// TwinCAT 3 PLC project PlcProject
// Title: Boikon Template
// Company: Boikon
// ProjectVersion: 0.7.1.0000
// ProgramVersion: 3.1.4026.23
// CompilerDefines: IsTemplate
// libraries:
//   [Boikon Library], * (Boikon)
//   CmpBitmapPool, * (System)
//   VisuDialogs, * (System)
//   VisuDialogs
// project tree:
//   / CHECKBOUNDS.TcPOU (excluded from build), GlobalTextList.TcGTLO, ImagePool.TcIPO (not stored), VisualizationManager.TcVMO (not stored)
//   DevelopmentPlayground/MurrModLight60/ cntrl_MurrModLight60.TcPOU, MurrModLight60_IO.TcDUT, eMurrModLight60Colors.TcDUT, MurrModLight60_Outputs.TcDUT
//   DevelopmentPlayground/ObjectOrientedExamples/ IOopExmpl.TcIO (excluded from build), OopExmplBase.TcPOU (excluded from build), OopExmplExtension.TcPOU (excluded from build), OopExmplMain.TcPOU (excluded from build), OopExmplRandomObjectWithInterface.TcPOU (excluded from build)
//   DevelopmentPlayground/UnitTesting/ BreakLogging.TcPOU, Vis_Test.TcVIS
//   General/HMI/ HMI_ERR_General.TcDUT, HMI_General.TcPOU, HMI_MAN_General.TcDUT, HMI_SP_General.TcDUT, HMI_SP_GeneralShared.TcDUT (not stored), HMI_STS_General.TcDUT, HMI_WRN_General.TcDUT (not stored)
//   General/ utl_General.TcPOU, Vis_General.TcVIS
//   Main/ MAIN.TcPOU, PlcTask.TcTTO, VisGeneral.TcVIS, VisScmTemplate.TcVIS
//   Version/ Global_Version.TcGVL
//   _Control_Templates/cntrl_RbtFanuc/ cntrl_RbtFanucUnloadingRobot.TcPOU
//   _Control_Templates/cntrl_RbtFanuc/HMI/ HMI_ERR_RbtFanucUnloading.TcDUT, HMI_MAN_RbtFanucUnloading.TcDUT, HMI_RbtFanucUnloading.TcPOU, HMI_SP_RbtFanucUnloading.TcDUT, HMI_STS_RbtFanucUnloading.TcDUT, HMI_WRN_RbtFanucUnloading.TcDUT, Vis_RbtFanucUnloading.TcVIS
//   _Control_Templates/cntrl_RbtFanuc/LinkedIO/ RbtFanucUnloading_DataIn.TcDUT, RbtFanucUnloading_DataOut.TcDUT
//   _Control_Templates/cntrl_RbtFanuc/LinkedIO/Helpers/ RbtFanucUnloading_Array8Uint.TcDUT, RbtFanucUnloading_DataIn_Grouped.TcDUT, RbtFanucUnloadingt_DataOut_Grouped.TcDUT, RbtFanucUnloading_DI.TcDUT, RbtFanucUnloading_DO.TcDUT, RbtFanucUnloading_GI.TcDUT, RbtFanucUnloading_GO.TcDUT
//   _Control_Templates/cntrl_SafetyController/ cntrl_SafetyController1.TcPOU, HMI_ERR_SafetyController1.TcDUT (not stored), HMI_SafetyController1.TcPOU, HMI_STS_SafetyController1.TcDUT (not stored), HMI_WRN_SafetyController1.TcDUT, Vis_SafetyZone1.TcVIS
//   _Control_Templates/ utl_SignalColumn.TcPOU
//   _Globals/ eLogGroupsProject.TcDUT, Glbl.TcGVL, Glcn.TcGVL
//   _Scam/SCM_TemplateClean/EnumsAndState/ eTpc.TcDUT, sTpc.TcPOU
//   _Scam/SCM_TemplateClean/HMI/ HMI_ERR_TemplateClean.TcDUT, HMI_MAN_TemplateClean.TcDUT, HMI_SP_TemplateClean.TcDUT, HMI_STS_TemplateClean.TcDUT, HMI_TemplateClean.TcPOU (not stored), HMI_WRN_TemplateClean.TcDUT (not stored)
//   _Scam/SCM_TemplateClean/ SCM_TemplateClean.TcPOU
//   _Scam/SCM_TemplateMachinePart/EnumsAndState/ eTMP.TcDUT, sTmp.TcPOU
//   _Scam/SCM_TemplateMachinePart/HMI/ HMI_ERR_TemplateMachinePart.TcDUT, HMI_MAN_TemplateMachinePart.TcDUT, HMI_SP_TemplateMachinePart.TcDUT (not stored), HMI_STS_TemplateMachinePart.TcDUT (not stored), HMI_TemplateMachinePart.TcPOU, HMI_WRN_TemplateMachinePart.TcDUT
//   _Scam/SCM_TemplateMachinePart/ SCM_TemplateMachinePart.TcPOU

CONFIGURATION PlcProject
    RESOURCE PLC ON TwinCAT3
        TASK PlcTask(INTERVAL := T#1ms, PRIORITY := 6);
        PROGRAM MAIN WITH PlcTask : MAIN;
    END_RESOURCE
END_CONFIGURATION

// ---- DevelopmentPlayground/MurrModLight60/MurrModLight60_IO.TcDUT
//ignore unused variables
{attribute 'analysis' := '-33'}
TYPE MurrModLight60_IO :
UNION
	//hw linking
	_Q AT %Q*: ARRAY[0..7] OF BYTE;
	//program use
	Control:MurrModLight60_Outputs;
END_UNION
END_TYPE

// ---- DevelopmentPlayground/MurrModLight60/eMurrModLight60Colors.TcDUT
{attribute 'qualified_only'}
{attribute 'strict'}
{attribute 'to_string'}
TYPE eMurrModLight60Colors :
(
	COLOR_OFF:= 		2#0,
	COLOR_RED:= 		2#001,
	COLOR_GREEN:= 		2#010,
	COLOR_YELLOW:= 		2#011,
	COLOR_BLUE:= 		2#100,
	COLOR_CUSTOM1:= 	2#101,
	COLOR_CUSTOM2:= 	2#110,
	COLOR_WHITE:= 		2#111,
	
	PAT_CONTINIOUS:= 	2#001000,
	PAT_BLINKING:=		2#010000,
	PAT_FLASHING:= 		2#011000,
	PAT_GRADBLINK:=		2#100000,
	
	SPD_LOW:=			2#01000000,
	SPD_MID:=			2#10000000,
	SPD_FAST:=			2#11000000
)BYTE;
END_TYPE

// ---- DevelopmentPlayground/MurrModLight60/MurrModLight60_Outputs.TcDUT
//ignore unused variables
{attribute 'analysis' := '-33'}
TYPE MurrModLight60_Outputs :
STRUCT
	//byte 0
	Stack1:BYTE; //combined bits for stack settings (color/pat/speed)
	//byte 1
	Stack2:BYTE; //combined bits for stack settings (color/pat/speed)
	//byte 2
	Stack3:BYTE; //combined bits for stack settings (color/pat/speed)
	
	//byte 3-4
	SpareByte3:BYTE;
	SpareByte4:BYTE;
	
	//byte 3
	BuzzerOnOff:BIT;
	BuzzerTypeBit0:BIT;
	BuzzerTypeBit1:BIT;
	BuzzerTypeBit2:BIT;

	BuzzerLoudnessBit0:BIT;
	BuzzerLoudnessBit1:BIT;
	BuzzerLoudnessBit2:BIT;
	BuzzerLoudnessBit3:BIT;
	
	//byte 4
	StackMode:BIT;
	LevelMode:BIT;
	SliceMode:BIT;
	SpareByte4_3:BIT;
	SyncModeAct:BIT;
	SyncModeTrig:BIT;
	UserPrefSelBit0:BIT;
	UserPrefSelBit1:BIT;
	
	//byte 5
	TopDown:BIT;
	SpareBYte5_1:BIT;
	ColorDom:BIT;
	EcoMode:BIT;
	SpareByte5_4:BIT;
	
	StacksBit0:BIT;		
	StacksBit1:BIT;
	StacksBit2:BIT;
END_STRUCT
END_TYPE

// ---- General/HMI/HMI_ERR_General.TcDUT
TYPE HMI_ERR_General :
STRUCT
	//General IO
	//prio's: emergency stop items == 100, e-circuit=99, default (nothing specified) = 50
	//adjust as needed
	ExampleErrorPreConfiggedPrio:BOOL;					//Error[prio=90] Example error with preconfigured prio (key only used at first creation/adding to the HMI-alarm-list-file)
END_STRUCT
END_TYPE

// ---- General/HMI/HMI_MAN_General.TcDUT
TYPE HMI_MAN_General :
STRUCT
	//note: manuals are normally used for controls, not for general
	//PB_MyManualCommand:bool;
END_STRUCT
END_TYPE

// ---- General/HMI/HMI_SP_General.TcDUT
TYPE HMI_SP_General :
STRUCT
	{warning 'TODO Template: example / remove when not needed'}
	//These setpoint are made available for all blocks
	Shared:HMI_SP_GeneralShared;											//Common setpoints used for multiple machine parts
END_STRUCT
END_TYPE

// ---- General/HMI/HMI_STS_General.TcDUT
TYPE HMI_STS_General :
STRUCT
	Version:STRING(23);								//Project version
END_STRUCT
END_TYPE

// ---- _Control_Templates/cntrl_RbtFanuc/HMI/HMI_ERR_RbtFanucUnloading.TcDUT
TYPE HMI_ERR_RbtFanucUnloading EXTENDS HMI_ERR_RbtFanuc:
STRUCT
	;//add custom bools on top of library block here
END_STRUCT
END_TYPE

// ---- _Control_Templates/cntrl_RbtFanuc/HMI/HMI_MAN_RbtFanucUnloading.TcDUT
TYPE HMI_MAN_RbtFanucUnloading EXTENDS HMI_MAN_RbtFanuc:
STRUCT
	;//add custom bools on top of library block here
END_STRUCT
END_TYPE

// ---- _Control_Templates/cntrl_RbtFanuc/HMI/HMI_SP_RbtFanucUnloading.TcDUT
TYPE HMI_SP_RbtFanucUnloading EXTENDS HMI_SP_RbtFanuc:
STRUCT
	;//add custom on top of library block here
END_STRUCT
END_TYPE

// ---- _Control_Templates/cntrl_RbtFanuc/HMI/HMI_STS_RbtFanucUnloading.TcDUT
TYPE HMI_STS_RbtFanucUnloading EXTENDS HMI_STS_RbtFanuc:
STRUCT
	;//add custom on top of library block here
END_STRUCT
END_TYPE

// ---- _Control_Templates/cntrl_RbtFanuc/HMI/HMI_WRN_RbtFanucUnloading.TcDUT
TYPE HMI_WRN_RbtFanucUnloading EXTENDS HMI_WRN_RbtFanuc:
STRUCT
	;//add custom bools on top of library block here
END_STRUCT
END_TYPE

// ---- _Control_Templates/cntrl_RbtFanuc/LinkedIO/RbtFanucUnloading_DataIn.TcDUT
{attribute 'analysis' := '-33'}
(*
	Plclinking:
		-Choose variable: ByAddress
			>
	Robot IO config:
		Go to config when you're in the DO/DI / UO/UI / GO/GI sections.
		if needed, delete default configs
		To link to ethercat card use, 
			rack 106 (some robot-types might use another rack nr. check manual) 
			slot 1
			start =>offset on the linked variables
			
		Example for this situation:
			UO => rack 106, slot 1, start 0   =>this will link UO[1]-CmdEnabled to ByAddress.0, which is good since Vars._UO.CmdEnabled is the first bit declared in the Vars structure.
			since the struct declared in the plc for the UO (Fanuc_StatusWord) is aligned to 3 bytes, DO must have an offset of 16
			DO => rack 106, slot 1, start 16 
*)
TYPE RbtFanucUnloading_DataIn :
UNION
	//linked directly to robot 
	ByAddress AT %I*: ARRAY[0..3] OF RbtFanucUnloading_Array8Uint;
	
	//data as variables for use in the plc
	Vars:RbtFanucUnloading_DataIn_Grouped;

END_UNION
END_TYPE

// ---- _Control_Templates/cntrl_RbtFanuc/LinkedIO/RbtFanucUnloading_DataOut.TcDUT
{attribute 'analysis' := '-33'}
(*
	Robot IO config:
		Go to config when you're in the DO/DI / UO/UI / GO/GI sections.
		if needed, delete default configs
		To link to ethercat card use, 
			rack 106 (some robot-types might use another rack nr. check manual) 
			slot 1
			start =>offset on the linked variables
			
		Example for this situation:
			UO => rack 106, slot 1, start 0   =>this will link UO[1]-CmdEnabled to ByAddress.0, which is good since Vars._UO.CmdEnabled is the first bit declared in the Vars structure.
			since the struct declared in the plc for the UO (Fanuc_StatusWord) is aligned to 3 bytes, DO must have an offset of 16
			DO => rack 106, slot 1, start 16 
*)
TYPE RbtFanucUnloading_DataOut :
UNION
	//linked directly to robot 
	ByAddress AT %Q*: ARRAY[0..3] OF RbtFanucUnloading_Array8Uint;
	
	//data as variables for use in the plc
	Vars:RbtFanucUnloadingt_DataOut_Grouped;

END_UNION
END_TYPE

// ---- _Control_Templates/cntrl_RbtFanuc/LinkedIO/Helpers/RbtFanucUnloading_Array8Uint.TcDUT
{attribute 'analysis' := '-33'}
TYPE RbtFanucUnloading_Array8Uint :
STRUCT
	_E: ARRAY [0..7] OF UINT;
END_STRUCT
END_TYPE

// ---- _Control_Templates/cntrl_RbtFanuc/LinkedIO/Helpers/RbtFanucUnloading_DataIn_Grouped.TcDUT
{attribute 'pack_mode' := '1'} //no gaps! (compiler tries to allign with base types)
TYPE RbtFanucUnloading_DataIn_Grouped :
STRUCT
	_UO:RbtFanuc_StatusWord; 			//24bits	>>start pt=1
	_DO:RbtFanucUnloading_DO;			//32 bits	>>start pt=25
	_GO:RbtFanucUnloading_GO;			//16 bits	>>start pt=57
END_STRUCT
END_TYPE

// ---- _Control_Templates/cntrl_RbtFanuc/LinkedIO/Helpers/RbtFanucUnloadingt_DataOut_Grouped.TcDUT
{attribute 'pack_mode' := '1'} //no gaps! (compiler tries to allign with base types and might skip bits otherwise)
{attribute 'analysis' := '-33'}
TYPE RbtFanucUnloadingt_DataOut_Grouped :
STRUCT
	_UI:RbtFanuc_ControlWord;			//24bits	>>start pt=1
	_DI:RbtFanucUnloading_DI;			//32 bits	>>start pt=25
	_GI:RbtFanucUnloading_GI;			//16 bits	>>start pt=57
END_STRUCT
END_TYPE

// ---- _Control_Templates/cntrl_RbtFanuc/LinkedIO/Helpers/RbtFanucUnloading_DI.TcDUT
{attribute 'analysis' := '-33'}
TYPE RbtFanucUnloading_DI :
STRUCT
	//bits 0-15
	SN_InitLeft:BIT;		//DI+00 command init/start left side
	SN_InitRight:BIT;		//DI+01 command init/start left side
	SN_CylInOk:BIT;			//DI+02 command resp cylinder is in
	SN_CylOutOk:BIT;		//DI+03 command resp cylinder is out
	SN_CrateEmptyOk:BIT;	//DI+04 command resp crate is empty
	SN_RequestDumpOk:BIT;	//DI+05 command resp crate is dumped
	SN_PayloadConfirm:BIT;	//DI+-6 command to confirm payload > must be setup in dcs
	bit07:BIT;
	bit08:BIT;
	bit09:BIT;
	PC_Left_Z:BIT;			//DI+10
	PC_Right_Z:BIT;			//DI+11
	PX_Left_X:BIT;			//DI+12
	PX_Right_X:BIT;			//DI+13
	bit14:BIT;
    bit15:BIT;
    K_DropBasket:BIT;		//Command from scam to drop basket
    bit17:BIT;
    bit18:BIT;
    bit19:BIT;
    bit20:BIT;
    bit21:BIT;
    bit22:BIT;
    bit23:BIT;
    bit24:BIT;
    bit25:BIT;
    bit26:BIT;
    bit27:BIT;
    bit28:BIT;
    bit29:BIT;
    bit30:BIT;
    bit31:BIT;
END_STRUCT
END_TYPE

(*
	//copy to your project and adapt names + number of bits to your situation
	//bits 0-15
	bit00:BIT;
    bit01:BIT;
    bit02:BIT;
    bit03:BIT;
    bit04:BIT;
    bit05:BIT;
    bit06:BIT;
    bit07:BIT;
    bit08:BIT;
    bit09:BIT;
    bit10:BIT;
    bit11:BIT;
    bit12:BIT;
    bit13:BIT;
    bit14:BIT;
    bit15:BIT;
    bit16:BIT;
    bit17:BIT;
    bit18:BIT;
    bit19:BIT;
    bit20:BIT;
    bit21:BIT;
    bit22:BIT;
    bit23:BIT;
    bit24:BIT;
    bit25:BIT;
    bit26:BIT;
    bit27:BIT;
    bit28:BIT;
    bit29:BIT;
    bit30:BIT;
    bit31:BIT;
*)

// ---- _Control_Templates/cntrl_RbtFanuc/LinkedIO/Helpers/RbtFanucUnloading_DO.TcDUT
{attribute 'analysis' := '-33'}
TYPE RbtFanucUnloading_DO :
STRUCT
	//bits 0-15
	SN_InitLeftOk:BIT;		//DO+00 command init/start left side
	SN_InitRightOk:BIT;		//DO+01 command init/start left side
	SN_CylIn:BIT;			//DO+02 command cylinder is in
	SN_CylOut:BIT;			//DO+03 command cylinder is out
	SN_CrateEmpty:BIT;		//DO+04 command crate is empty
	SN_RequestDump:BIT;		//DO+05 command crate is dumped
    bit06:BIT;
    bit07:BIT;
    bit08:BIT;
	STS_Error:BIT;			//DO+09 status in error
    STS_Latched1:BIT;		//DO+10
    STS_Latched2:BIT;		//DO+11
    bit12:BIT;
    bit13:BIT;
    bit14:BIT;
    bit15:BIT;
	K_DropBasket_OK:BIT;	//Response from robot drop basket ok
    bit17:BIT;
    bit18:BIT;
    bit19:BIT;
    bit20:BIT;
    bit21:BIT;
    bit22:BIT;
    bit23:BIT;
    bit24:BIT;
    bit25:BIT;
    bit26:BIT;
    bit27:BIT;
    bit28:BIT;
    bit29:BIT;
    bit30:BIT;
    bit31:BIT;
END_STRUCT
END_TYPE


(*
bit00:BIT;
    bit01:BIT;
    bit02:BIT;
    bit03:BIT;
    bit04:BIT;
    bit05:BIT;
    bit06:BIT;
    bit07:BIT;
    bit08:BIT;
    bit09:BIT;
    bit10:BIT;
    bit11:BIT;
    bit12:BIT;
    bit13:BIT;
    bit14:BIT;
    bit15:BIT;
    bit16:BIT;
    bit17:BIT;
    bit18:BIT;
    bit19:BIT;
    bit20:BIT;
    bit21:BIT;
    bit22:BIT;
    bit23:BIT;
    bit24:BIT;
    bit25:BIT;
    bit26:BIT;
    bit27:BIT;
    bit28:BIT;
    bit29:BIT;
    bit30:BIT;
    bit31:BIT;
*)

// ---- _Control_Templates/cntrl_RbtFanuc/LinkedIO/Helpers/RbtFanucUnloading_GI.TcDUT
{attribute 'analysis' := '-33'}
TYPE RbtFanucUnloading_GI :
STRUCT
	//copy to your project and adapt names + number of bits to your situation
	Word0:WORD;
END_STRUCT
END_TYPE

// ---- _Control_Templates/cntrl_RbtFanuc/LinkedIO/Helpers/RbtFanucUnloading_GO.TcDUT
{attribute 'analysis' := '-33'}
TYPE RbtFanucUnloading_GO :
STRUCT
	//GO[1]
	ErrorNr:UINT;
	State:UINT;
	NrPickedCrates:UINT;
	NrPayload:uint;
END_STRUCT
END_TYPE

// ---- _Control_Templates/cntrl_SafetyController/HMI_WRN_SafetyController1.TcDUT
//Extend the base errors with project errors
TYPE HMI_WRN_SafetyController1 EXTENDS HMI_WRN_SafetyLogic:
STRUCT
	//note: errors for inputs moved to input-instances
	;
END_STRUCT
END_TYPE

// ---- _Globals/eLogGroupsProject.TcDUT
{attribute 'qualified_only'}
TYPE eLogGroupsProject :
(
	//the first 8 bits are taken/reserved for the boikon library groups: Boikon_Library.eLogGroups
	(*
	Off					:= 2#0,					//this channel will not get logged
	Default				:= 2#1,					//the library blocks will automaticly give the default group for the logged type, otherwise a custom group can be chosen
	Inputs				:= 2#10,	
	Outputs 			:= 2#100,
	Analogs				:= 2#1000,
	Cntrl_states		:= 2#10000,				//states for controls/utilities (servo blocks for example)
	*)
	//project groups, in total 32 bits available
	//add/rename/remove groups as needed
	SCM_States 			:=SHL(2#1,8),
	SCM_CommSignals		:=SHL(2#1,9),
	Spare				:=SHL(2#1,10),
	Template			:=SHL(2#1,11),
	TestServoPos		:=SHL(2#1,12)
)DWORD;
END_TYPE

//info on attributes:
//strict 			: also tests if the name is not used for something else
//to_string			: allows the enum to be converted to string
//qualified_only 	: forces the user to start witht the type name (to avoid the situation that accidentially another enum is used)

// ---- _Scam/SCM_TemplateClean/EnumsAndState/eTpc.TcDUT
//enum of states
{attribute 'strict'}
{attribute 'to_string'}
{attribute 'qualified_only'}
TYPE eTpc :
(
	//NOTE @ copy of this enum, adapt existing state names:
	Disabled := -1, //-1: to make sure the code for disabling fires
	TotalReset,
	Initialise,
	Rest
)INT;
END_TYPE

//info on attributes:
//strict 			: don't allow mixing of types
//to_string			: allows the enum to be converted to string
//qualified_only 	: forces the user to start witht the type name (to avoid the situation that accidentially another enum is used)

// ---- _Scam/SCM_TemplateClean/HMI/HMI_ERR_TemplateClean.TcDUT
TYPE HMI_ERR_TemplateClean :
STRUCT
	(*
		Rules:
		Errors shall only be off type BOOL
		Errors shall be set >> the HMI block will do the resetting

		Syntax convention:
		a clear variable name which describes the error			as described below
		InitNotEmpty:BOOL;										//Error [machinepart]: not empty during initialisation
		
		prio's: emergency stop items == 100, e-circuit=99, default (nothing specified) = 50
		adjust as needed
		//example how to pre-set error priorities for the HMI. Default errors get prio 50, Recommend prio 100 for e-stop buttons etc
		ExampleErrorPreConfiggedPrio:BOOL;					//Error[prio=90] Example error with preconfigured prio (key only used at first creation/adding to the HMI-alarm-list-file)
	*)
END_STRUCT
END_TYPE

// ---- _Scam/SCM_TemplateClean/HMI/HMI_MAN_TemplateClean.TcDUT
TYPE HMI_MAN_TemplateClean :
STRUCT

END_STRUCT
END_TYPE

// ---- _Scam/SCM_TemplateClean/HMI/HMI_SP_TemplateClean.TcDUT
TYPE HMI_SP_TemplateClean :
STRUCT
	MachinePartEnabled:BOOL:=TRUE;				//block is enabled >> can be used to disable part(s) of the machine
END_STRUCT
END_TYPE

// ---- _Scam/SCM_TemplateClean/HMI/HMI_STS_TemplateClean.TcDUT
TYPE HMI_STS_TemplateClean :
STRUCT
	IsEmpty:BOOL;												//Machinepart is empty
END_STRUCT
END_TYPE

// ---- _Scam/SCM_TemplateMachinePart/EnumsAndState/eTMP.TcDUT
//enum of states
{attribute 'strict'}
{attribute 'to_string'}
{attribute 'qualified_only'}
TYPE eTMP :
(
	TotalReset,
	InitCyl,
	InitSrv,
	InitCamQuickFocus,
	InitCamLoadJob,
	Rest,
	SrvPosStart,
	SrvPosStartInterl,
	SrvPosEnd,
	SrvPosEndIntrl,
	CylOut,
	CylIn,
	MtrStartFwd,
	MtrStop,
	MtrStartRev,
	CamReady,
	CamTrig,
	MultiStepTest2,
	MultiStepTest3,
	
	//Example how to use the organiser semi-automode
	//this is a special case in which the operator can choose with a button for example to let the machine do special things 
	//like put servos+clinders automated in a position for configuring/measuring
	
	SemiAutoStart,
	SemiAutoStop
);
END_TYPE

//info on attributes:
//strict 			: don't allow mixing of types
//to_string			: allows the enum to be converted to string
//qualified_only 	: forces the user to start witht the type name (to avoid the situation that accidentially another enum is used)

// ---- _Scam/SCM_TemplateMachinePart/HMI/HMI_ERR_TemplateMachinePart.TcDUT
TYPE HMI_ERR_TemplateMachinePart :
STRUCT
	(*
		Rules:
		Errors shall only be off type BOOL
		Errors shall be set >> the HMI block will do the resetting

		Syntax convention:
		a clear variable name which describes the error			as described below
		InitNotEmpty:BOOL;										//Error [machinepart]: not empty during initialisation
		
		prio's: emergency stop items == 100, e-circuit=99, default (nothing specified) = 50
		adjust as needed
		//example how to pre-set error priorities for the HMI. Default errors get prio 50, Recommend prio 100 for e-stop buttons etc
		ExampleAddPrioForHmiError:BOOL;					//Error[prio=90] TemplateMachinePart: we have an error!
	*)
	InitNotEmpty:BOOL;								//Error [machinepart]: not empty during initialisation
	
	//example how to pre-set error priorities for the HMI. Default errors get prio 50, Recommend prio 100 for e-stop buttons etc
	ExampleAddPrioForHmiError:BOOL;					//Error[prio=100] TemplateMachinePart: we have an error!
	
	//test log error by name, very long name, truncation
	TestStupidLongErrorNameWillItGetLoggedAbcdefghijklmnopqrstuvwzyzAbcdefghijklmnopqrstuvwzyzAbcdefghijklmnopqrstuvwzyzAbcdefghijklmnopqrstuvwzyzAbcdefghijklmnopqrstuvwzyz:BOOL;
END_STRUCT
END_TYPE

// ---- _Scam/SCM_TemplateMachinePart/HMI/HMI_MAN_TemplateMachinePart.TcDUT
TYPE HMI_MAN_TemplateMachinePart :
STRUCT
	;
END_STRUCT
END_TYPE

// ---- _Scam/SCM_TemplateMachinePart/HMI/HMI_WRN_TemplateMachinePart.TcDUT
TYPE HMI_WRN_TemplateMachinePart :
STRUCT
	(*
		Rules:
		Warnings shall only be of type BOOL
		Warnings can be set / reset / activated as you need it (unlike errors!). 
		
		Syntax convention:
		a clear variable name which describes the warning		as described below
		StepLockActive:BOOL;									//Warning [machinepart]: in step modus (steps are held until confirmation the continue to the next step)
	*)
	NotRdyRcv_Discharge:BOOL;								//Warning [machinepart]: not ready to receive products
	CameraNotReady:BOOL;									//Warning [machinepart]: waiting for camera ready
	PlanoBufferNeedsRefill:BOOL;							//Warning [machinepart]: Planobuffer needs refill
END_STRUCT
END_TYPE

// ---- Version/Global_Version.TcGVL
{attribute 'TcGenerated'}
{attribute 'no-analysis'}
{attribute 'linkalways'}
// This function has been automatically generated from the project information.
VAR_GLOBAL CONSTANT
	{attribute 'const_non_replaced'}
	stLibVersion_Boikon_Template : ST_LibVersion := (iMajor := 0, iMinor := 7, iBuild := 1, iRevision := 0, nFlags := 0, sVersion := '0.7.1.0');
END_VAR

// ---- _Globals/Glbl.TcGVL
//project related global variables
{attribute 'qualified_only'}
{attribute 'analysis' := '-33'}
VAR_GLOBAL
//Variables set by Checkbounds. This function increases processor load and should be disabled once bounds problems are solved
	OutOfBounds:BOOL:=FALSE;						//Should always be false otherwise a bounds problem >> function CHECKBOUNDS must be implemented in the project, check the beckhoff help !only for testing purposes!
	OutOfBoundsIndex:DINT := 0;						//Index trying to address which was out of bounds


(*Project*)
	//TODO TEMPLATE >>
		//adapt / remove as needed
	SimEnable:BOOL:=FALSE;					//Enable simulation (when false, all simulation setpoints will be set to false
	Sim_MyMachinePart:BOOL; 				//Simulate only a part of the machine (in this case the template example)
END_VAR
// {attribute 'qualified_only'} >>forces the user to add the DUT name in front of the variables
// {attribute 'analysis' := '-33'} >>deactivate error unused variable for next variable/struct

// ---- _Globals/Glcn.TcGVL
//project related global constants
{attribute 'qualified_only'}
VAR_GLOBAL CONSTANT

{info 'TODO: TEMPLATE REMOVE WHEN NOT NEEDED'}
//array sizes >> use this to initialise the array AND then use it in the for loops which run through the arrays etc
	//MaxIndexForMyArray:INT:=10;
	//to be used as:
	//MyArray: array[0..MaxIndexForMyArray] of bool;
	//and then
	//FOR index:=0 to MaxIndexForMyArray by 1 DO ...
END_VAR

// ---- DevelopmentPlayground/ObjectOrientedExamples/IOopExmpl.TcIO
(*An interface describes the must have methods for a functionblock
	-now you know for sure that a block implementing this interface will have the methods described here
*) 
INTERFACE IOopExmpl

METHOD MustHaveMethod : BOOL
VAR_INPUT
	I:BOOL;
END_VAR
END_METHOD

END_INTERFACE

// ---- Main/MAIN.TcPOU
(*Basic MAIN with an example organiser and scam*)
{info '_Welcome to the Boikon Twincat 3 Template'}
{info '__Please read the _Readme.txt for more info'}
{warning 'TODO Template: upload boot project at online change is disabled in project settings, RE-ENABLE!!!!'}
PROGRAM MAIN
VAR
	//General collection of system wide IO and control blocks
	General: Utl_General;

	//TODO TEMPLATE: here in the example only 1 organiser is used, add + rename as needed
	Organiser:cntrl_Organiser(						
		SP_TmrReset := T#1S,
		SP_TmrResetES := T#3S);
END_VAR

//TODO TEMPLATE >> Remove this section, it is for testing the library and template
//Also remove the define from here: project/properties/compile/compiler defines/IsTemplate
{IF defined (IsTemplate)}
	{warning 'TODO Template: testing is enabled >> Remove the define and clean all "TODO TEMPLATE" locations'}
	{attribute 'analysis' := '-33'}
	VAR
		//Scam-template >> use tool supplied in the folder, to make a copy for your own scam implementation 
		OrganiserFake: cntrl_OrganiserFake;
		
		//Fully functional test scam which uses almost all library blocks >> can be used as example how to do things 
		ExampleMachinePart: SCM_TemplateClean;

		//just to show it's possible
		//these variables will now have the same comment (these 2 lines)
		//*multiline comment still is a kind of broken in the editor, parts will dissapear..
		MyBool1,MyBool2,MyBool3:BOOL;  

		//Banner-Multicolor signal lamp
		//NOTE: You can use it this way for multiple organisers as well, just keep calling ..M_UpdateOrganiserState(xxx) for each organiser  
		LP_OrgGroupMachinePart:Cntrl_BannerKxx(
			Intensity:= eBannerKxx_Intensity.Low);

		LP_MurrTest: cntrl_MurrModLight60(NrOfStacks:=3);

		//Performance test	
		HM_ProfileBlocks:BOOL;
		StopWatchGeneral,StopWatchMachineStuff:profiler;
		
		//casting works with a lot of types, example time
		sMyUtcTime:string;

		//string value to int test
		sValue1,sValue2,sValue3:STRING := '123';
		sValue4,sValue5:string(1);
		b0Value:BYTE;
		iValue1,iValue2:INT;
		
		
		//random tests
		dbglreal:LREAL;
		dbgbool1,dbgbool2,dbgbool3:BOOL;
	END_VAR
{END_IF}

//TODO template: general actions can be added here. 
//in utl_General I've added the usual suspects needed for a machine.
//please keep in mind I've only included common reocurring items, you need to thoroughly check / update / clean the block!
a_General();
b_MachinePart();

ACTION a_General:
//General is the place for all in-/outputs not specific belonging to a machinepart like:
//	-handling of boikonlibrary functionality
//	-general start/stop/reset buttons + lights
//	-general airpressure sensor
//	-safety components: control + errors for doors/lightscreens/pushbuttons
//	-ethercat diagnostics
General(
	//Reset command + general start/stop/reset button lights > add organisers as needed, use OR
	I_SN_ResetErrors:= Organiser.Reset_K,
	I_SN_Lp_Pb_StartAll:= Organiser.Q_LP_Start,
	I_SN_Lp_Pb_StopAll:= Organiser.Q_LP_Stop,
	I_SN_Lp_Pb_ResetAll:= Organiser.Q_LP_Reset,
	
	//Machine status
	I_STS_Error:=,
	I_STS_NoDischarge:=,
	I_STS_OperatorInput:=,
	I_STS_Running:=,	
	
	//Organiser/SCAM control-outputs
	Q_SN_ES_Zone1_OK=>, 
	Q_SN_StartAll=>,
	Q_SN_StopAll=>,
	Q_SN_ResetAll=> ,
	Q_SN_TotalResetAll=>);

//TODO TEMPLATE remove if not needed
//Organiser(s) Banner multicolor indicator light
//	this is an example on how to use it to show the status of an organiser
//	1) you can also manually control the lamp with the given M_Set... methods, but then don't call M_UpdateOrganiserState anymore!
//	2) inside general would be a better place but there you can't access the Organiser instances easily (or you tresspass OOP by doing things like: main.Organiser inside.... > don't do that!)
LP_OrgGroupMachinePart.M_UpdateOrganiserState(Organiser); //call this method for each organiser belonging to this group
LP_OrgGroupMachinePart();

//TODO TEMPLATE remove banner break-time
//Mess around with the banner multicolor lamp >> if break-time, overwrite previous (organiser-state) call with a manual set color
IF(	(	BknGlbl.LocalSystemTime.wHour = 10
		AND_THEN BknGlbl.LocalSystemTime.wMinute <= 15)
	OR	(	BknGlbl.LocalSystemTime.wHour = 12
			AND_THEN BknGlbl.LocalSystemTime.wMinute >= 30)
	OR	(	BknGlbl.LocalSystemTime.wHour >= 17))
THEN
	LP_OrgGroupMachinePart.M_Set2ColorAnimation(
		I_Color1 := eBannerKxx_Color.Yellow,
		I_Color2 := eBannerKxx_Color.Red,
		I_Animation:= eBannerKxx_AnimationType.HalfHalfRotate,
		TRUE); 
	LP_OrgGroupMachinePart();
END_IF
END_ACTION

ACTION b_MachinePart:
//Note: if the machine consists of several machine parts with their own organiser then for a cleaner structure make a seperate action for each part
//todo think about this

Organiser(
	//Emergencystop zone for scams connected to this organiser
	I_SN_ES_OK:= General.Q_SN_ES_Zone1_OK,
	I_SN_ExternalError:= General.Q_SN_ERR_General, //organiser should go into error caused by external factors (like a general error)
	//Total reset command for this organiser and connected scams
	//note: scams that communicate with each other via interlocking should have the same total reset command otherwise deadlocks will occur!
	I_SN_TotalReset:= General.Q_SN_TotalResetAll,
	I_PB_Start:= General.Q_SN_StartAll,
	I_PB_Stop:= General.Q_SN_StopAll,
	I_PB_Reset:= General.Q_SN_ResetAll, 
	Q_LP_Start=>, 
	Q_LP_Stop=>, 
	Q_LP_Reset=>);

ExampleMachinePart( //todo remove true
	I_K_ES_OK:= General.Q_SN_ES_Zone1_OK, 			//Emergency stop for this zone OK. @ mutliple zones, fbGeneral must be adapted to supply these signals for each zone
	I_Organiser:= Organiser, 						//Control signals from the organiser
	I_STS_SUP_Empty:= , 							//Connect to upstream. The upstream is empty, use this to enter energy-save mode (stop conveyors etc)
	Q_STS_Empty=> , 								//Connect to downstream. The supply is empty and this part is now empty and in energy-save mode
	Q_SN_SUP_Request=> ,							//Connect to upstream. This program is running and ready to receive products
);
END_ACTION

END_PROGRAM

// ---- General/utl_General.TcPOU
(* 	General I/O handling 

	TODO TEMPLATE INFO:
		This is a template for handling of general actions. It should cover your basic needs.
		I've included actions that I commonly needed in my projects but keep in mind this whole block is a suggestion and needs to be updated to your project needs!
		Over time, more and more got included in the boikonlibrary so this block gets cleaner.
		
		Changes that might be needed:
		*As the block is now, it is assumed that with a set of general buttons everything needs to be started >> I_PB_xxxx inputs. Change to your projects needs
		*If your machine is divided into multiple subsections which have their own buttons / safety zones then I recommend to:
			-make unique general fb's per section.
				*General  				>calls the boikon library and handles stuff that is needed for all sections (if there are no xxx_all buttons than remove them here)
				*General_ZoneX			>handles buttons / safety zone for this section (does NOT call the boikonLibrary! that should only be done once)
				*...
		-I've added a TotalResetAll output to this general, the idea is that sometimes you need all organisers to be total reset at once. 
		Especially if blocks are communicating with each other with interlocks this is needed (for those to be total reset together). 
		In that case use this signal for those organisers + Hide the total reset button for these organisers in the HMI (the organiser viewscreen has a property for this) so the single organiser total reset can't be done.

	Usage:
		Use Q_SN_Start/Stop/Reset/TotalReset-All signals for the organisers that should be started whith the buttons defined here
		Use Q_SN_ES_Zone1_OK for the scams that belong to this zone
		Use Q_SN_ERR_General for the organisers (high if 1 of the errors defined here is set >>safety/air/ups/...)
*)
FUNCTION_BLOCK utl_General;
VAR_INPUT
	I_SN_ResetErrors:BOOL;						//Signal reset general errors
	I_SN_Lp_Pb_StartAll:BOOL;					//Signal activate lamp pushbutton >> if only 1 organiser, connect directly to specific organiser output, in case of multiple organisers make it sensible yourself
	I_SN_Lp_Pb_StopAll:BOOL;					//Signal activate lamp pushbutton >> if only 1 organiser, connect directly to specific organiser output, in case of multiple organisers make it sensible yourself
	I_SN_Lp_Pb_ResetAll:BOOL;					//Signal activate lamp pushbutton >> if only 1 organiser, connect directly to specific organiser output, in case of multiple organisers make it sensible yourself
	
	//Machine status (used for signal column)
	I_STS_Error:BOOL;							//Status any machine-part is in error (any organiser in error state)
	I_STS_Running:BOOL;							//Status all machine-parts are running (all organisers in Auto_K)
	I_STS_NoDischarge:BOOL;						//Status discharge (next machine) not accepting products
	I_STS_OperatorInput:BOOL;					//Status any machine-part needs operator interaction
END_VAR

VAR_OUTPUT
	Q_SN_ES_Zone1_OK:BOOL;						//Signal general emergency stop circuit is OK
	Q_SN_ERR_General:BOOL;						//Signal general error >> use to put organisers in state error
	
	Q_SN_StartAll:BOOL;							//Signal FOR all machine parts pushbutton is pressed
	Q_SN_StopAll:BOOL;							//Signal FOR all machine parts pushbutton is pressed
	Q_SN_ResetAll:BOOL;							//Signal FOR all machine parts pushbutton is pressed
	Q_SN_TotalResetAll:BOOL;
END_VAR

VAR
(*Configuration*)	

(*Logged variables*)

(*Internals*)

(*Instances*)
	HMI:HMI_General;						//All HMI related variables
	OrganiserGeneral:cntrl_OrganiserFake;	//Fake organiser for HMI reset signals etc
	GetCurrentTaskInfo:GETCURTASKINDEX;		//Get plc task information
	PbSf_TotalResetAll:utl_PB_HmiSafe;		//Pushbutton-safe for HMI totalreset button >> total reset all programs of this safety zone (connect to correct organisers!)
	BknLibrary:utl_BknLibrary(				//Handles library functionality (BknGlb-variables + logging)
		EnableTaskCycleTimeExceedWarning:=TRUE);			//dis/enable cycletime exceeding warnings (you really shouldn't...)

	//TODO TEMPLATE >> This is a template block which uses the boikon default. You might have to adapt this block based on the customers requirements
	SignalColumn: utl_SignalColumn;

	//TODO TEMPLATE >>
		//Remove if you don't have a cx2100-xxx module
		//Configure correctly if it has an ups and set the correct address (hw-config, second tab esb-device)
		//NOTE: with button ENTER it will show the ip address of the first adapter then with UP/DOWN you can cycle through the adapters
		//twincat on BSD>> before it worked I had to "disable virtual device names" in the hw-config for the usb host device
	CxPowerSupply: cntrl_CxPowerSupply(
					Options:= 0,
					CxAddress:= 16#7004);

	//TODO TEMPLATE >> 
		//Make 1 instance per ethercat master
		//per ethercat master device:
		//Link "I_AmsNetID" to the master ethercat device. If this is not linked, then the block is disabled.
		//if you need delayed auto start of the ethercat master then make this setting in the hw-config:
		//	master device/ethercat/advanced settings/state machine/master settings/startup state >> set to init
	EthercatManager:cntrl_EthercatManager(DelayedStartMaster:= TRUE);	//Ethercat devices manager
	
	//TODO TEMPLATE 
		//>> adapt safety template as needed + rename
		//>> the template example controls multiple groups but if you want you can create a controller/group	
	SafetyController:cntrl_SafetyController1; //note: this block extends the basic mandatory functionality. The extension (located in your project) has to be adapted as needed
	
	//TODO TEMPLATE 
		//make syncunits for groups of terminals which belongs together (all terminals behind a EK1122)
		//make an instance per syncunit here and hw-link to the wc-state of the syncunit group 
	I_WcState_MCC: cntrl_SyncUnitMonitor;			//SyncUnitGroup for main cabinet 
	I_WcState_RIO1: cntrl_SyncUnitMonitor;			//SyncUnitGroup for RIO1
	I_WcState_SafetyZones: cntrl_SyncUnitMonitor;	//SyncUnitGroup for safety
	

	I_PS_AirpressureOk: cntrl_InputHmiStsErr;		//Pressure switch airpressure ok 
	I_UPS_InBatteryMode: cntrl_InputHmiStsErr;		//UPS running on battery
	I_Pb_StartAll: cntrl_Input;						//Pushbutton start that should start the whole machine. If a machine has different zones, then create per zone a general >> example djura subs
	I_PbNc_StopAll:cntrl_Input;						//Pushbutton stop normally closed that should start the whole machine. If a machine has different zones, then create per zone a general >> example djura subs
	I_Pb_ResetAll: cntrl_Input;						//Pushbutton reset that should start the whole machine. IF a machine has different zones, THEN create per zone a general >> example djura subs
	
	
(*Inputs / Outputs*)	
	Q_Lp_StartAll AT %Q*:BOOL; 						//Lamp pushbutton start whole machine
	Q_Lp_StopAll AT %Q*:BOOL; 						//Lamp pushbutton stop whole machine
	Q_Lp_ResetAll AT %Q*:BOOL; 						//Lamp pushbutton reset whole machine
	
END_VAR

(*All HMI related thingies: Errors/Warnings/Statusses/etc*)
_M_HMI();

(*Simulation*)
A_Simulation();

(*Global variables, must run first (detection first scan)*)
A_Globals();

(*Outputs / Signals / Globals / etc*)
A_Activations();

METHOD PRIVATE _M_HMI
//Update HMI variables (check error status + reset, check warnings)
HMI.M_Update(	I_OrgControl:= OrganiserGeneral,
				I_HMI_Parent := 0, 				//This is top level, no error propagation
				I_ERR:= HMI.ERR,
				I_WRN:= HMI.WRN,
				I_MAN:= HMI.MAN);
		
//Statusses
	
//Warnings
HMI.WRN.CheckBoundsTriggered := Glbl.OutOfBounds;

//Errors
HMI.ERR.ExampleErrorPreConfiggedPrio s= BknGlbl.FirstScan;
END_METHOD

ACTION A_Activations:
//Signals 
Q_SN_ERR_General := HMI.P_STS_InError;

Q_SN_ES_Zone1_OK := SafetyController.Q_K_ES_Zone1_OK; 

Q_SN_StartAll := I_Pb_StartAll.Q;
					
Q_SN_StopAll := NOT I_PbNc_StopAll.Q;

Q_SN_ResetAll := 	I_Pb_ResetAll.Q; 
					//DO NOT ADD: I_SN_ResetErrors    
						//ELSE a reset loop will happen (linked to organiser(s), org reset linked back to general)

Q_SN_TotalResetAll := (	.BknGlbl.FirstScan
						OR PbSf_TotalResetAll.Q);

(*Outputs*)
Q_Lp_StartAll := 	I_SN_Lp_Pb_StartAll;
Q_Lp_StopAll := 	I_SN_Lp_Pb_StopAll;
Q_Lp_ResetAll := 	I_SN_Lp_Pb_ResetAll
					OR Q_SN_ERR_General;

//TODO TEMPLATE
	//If your machine has only 1 organiser OR you have a seperate organiser for each machine part then you can consider using "real" organisers in here (remove this fake organiser in that case)
//Fake organiser >> handles reset signals + logging. Is extra needed because the controls declared in general need this variable's interface
OrganiserGeneral(	I_K_Reset:= I_SN_ResetErrors OR Q_SN_ResetAll, 
					I_K_Auto:= FALSE);
			
//Boikon library funtionality   
GetCurrentTaskInfo();
BknLibrary(
	I_HMI_Parent:= HMI, 
	I_OrgControl:= OrganiserGeneral,
	IO_TaskInfo:= _TaskInfo[GetCurrentTaskInfo.Index],
	IO_AppInfo:= _AppInfo);

//Machine status signal column	
SignalColumn(
	I_STS_Error:= I_STS_Error , 
	I_STS_Running:= I_STS_Running, 
	I_STS_NoDischarge:= I_STS_NoDischarge, 
	I_STS_OperatorInput:= I_STS_OperatorInput);
	
//TODO TEMPLATE see instructions @ declaration
CxPowerSupply(
	I_HMI_Parent:= HMI,
	I_OrgControl:= OrganiserGeneral,
	I_K_SimulationActive:= Glbl.SimEnable);

//TODO TEMPLATE see instructions @ declaration
//Ethercatdevice managers
EthercatManager(
	Q_STS_NrOfSlavesNotInOp=>);

//TODO TEMPLATE >> see instructions @ instance declaration and comment inside this block
	//note: nicest way to restart safety is to use a dedicated hw button. Here I've connected it to the more general reset signal/buttons
SafetyController(
	I_HMI_Parent:= HMI,
	I_K_SimulationActive:= 	Glbl.SimEnable,		//TODO TEMPLATE >> remove this line (for unittesting I've a "real" safety setup on the testboard that manipulates safety card inputs with plc output)
	I_K_Enable:= I_WcState_SafetyZones.Q_STS_SyncUnitDataOk, 			//NOTE: connecting enable like this has the advantage that safety is started and ErrAcked at startup of ethercat
																		//Disadvantage is that it will auto reset errors at restart of ethercat (you might find this an advantage...)
	I_OrgControl:= OrganiserGeneral,
	I_STS_AirPressure_OK := I_PS_AirpressureOk.Q);

//cntrl_Inputs need to be called cyclically
I_Pb_StartAll(
	I_K_SimulationActive:= Glbl.SimEnable, 
	//I_K_SimulateOn:= , >>overwritten by visu general 
	);

//RE > preset sim-on
I_PbNc_StopAll.I_K_SimulateOn S= Glbl.SimEnable AND NOT I_PbNc_StopAll.I_K_SimulationActive;
I_PbNc_StopAll(
	I_K_SimulationActive:= Glbl.SimEnable, 
	//I_K_SimulateOn:= , >>overwritten by visu general 
	);
	
I_Pb_ResetAll(
	I_K_SimulationActive:= Glbl.SimEnable, 
	//I_K_SimulateOn:= , >>overwritten by visu general 
	);

//safebuttons need to be called cyclically
PbSf_TotalResetAll();
	
//General statusses
//TODO TEMPLATE >> read comment @ instance declaration 
I_WcState_MCC(
	I_HMI_Parent:= HMI,
	I_OrgControl:= OrganiserGeneral,
	I_K_SimulationActive:= Glbl.SimEnable, 
	I_K_SimulateDataValid:= TRUE);

I_WcState_RIO1(
	I_HMI_Parent:= HMI,
	I_OrgControl:= OrganiserGeneral,
	I_K_SimulationActive:= Glbl.SimEnable, 
	I_K_SimulateDataValid:= TRUE);
				
I_WcState_SafetyZones(
	I_HMI_Parent:= HMI,
	I_OrgControl:= OrganiserGeneral,
	I_K_SimulationActive:= Glbl.SimEnable, 
	I_K_SimulateDataValid:= TRUE);
	
I_PS_AirpressureOk(
	I_HMI_Parent := HMI,
	I_OrgControl := OrganiserGeneral,
	I_K_SetError := NOT I_PS_AirpressureOk.Q,
	I_K_SimulationActive:= Glbl.SimEnable, //TODO TEMPLATE, remove OR UnitTesting
	I_K_SimulateOn:= TRUE);

//TODO TEMPLATE >> dependant on your ups solution adapt as needed
I_UPS_InBatteryMode(
	I_HMI_Parent := HMI,
	I_OrgControl := OrganiserGeneral,
	I_K_SetError := I_UPS_InBatteryMode.Q,
	I_K_SimulationActive:= Glbl.SimEnable, 
	I_K_SimulateOn:= FALSE);
END_ACTION

ACTION A_Globals:
//if firstscan or program changed >> ...
IF(	BknGlbl.FirstScan
	OR BknGlbl.FirstScanOnlineChange)
THEN
	//current project version >> autogenerated, sometimes autogenerator takes a second build before the file is generated
	{IF defined (variable:stLibVersion_Boikon_Template)}
		HMI.STS.Version := Global_Version.stLibVersion_Boikon_Template.sVersion;
	{ELSE}
		HMI.STS.Version := 'Needs Fixing';
	{END_IF}
	//reset out of bounds detection
	Glbl.OutOfBounds := FALSE;
END_IF
END_ACTION

ACTION A_Simulation:
//TODO Template >> adapt as needed

//if simulation not enabled or firstscan detected >> reset all simulations
IF(	NOT Glbl.SimEnable
	OR BknGlbl.FirstScan)
THEN
	Glbl.SimEnable := FALSE;
END_IF
END_ACTION

{attribute 'suppress_wrn_C0410'} //oh nooo... the number in the warning is c5410 but this is how you disable it????
PROPERTY P_SP_Shared : REFERENCE TO HMI_SP_GeneralShared
GET
P_SP_Shared REF= HMI.SP.Shared;
END_GET
END_PROPERTY

END_FUNCTION_BLOCK

// ---- General/HMI/HMI_General.TcPOU
(*	HMI variables

	This block holds all HMI variables and handles communication with the HMI
	
	2024-02 HP
		-initial
*)
{attribute 'no_explicit_call' := 'do not call this POU directly'}
FUNCTION_BLOCK HMI_General EXTENDS HMI_BaseBlock

//HMI variables that can be written to by the plc and HMI 
VAR_INPUT
	//Do not change these names, the HMI is hardcoded to use these exact names
	MAN:HMI_MAN_General;				//HMI manuals
	STS:HMI_STS_General;				//HMI statusses
	WRN:HMI_WRN_General;				//HMI warnings
	ERR:HMI_ERR_General;				//HMI errors
END_VAR

//Hmi variables that can only be written to by the HMI and read by the plc
VAR_OUTPUT PERSISTENT
	//Do not change these names, the HMI is hardcoded to use these exact names
	SP:HMI_SP_General;					//HMI setpoints
END_VAR

//this block should not be called

END_FUNCTION_BLOCK

// ---- _Control_Templates/utl_SignalColumn.TcPOU
(* Signal column with default (BOIKON) colors

	This block is the boikon default for a signal column.
	Per customer it may vary how to colors have to work, this is why this block is in the project and not in the library
		>Adapt as needed!
	
	Changes
	2025-10-09
		-it's alive
	
*)

FUNCTION_BLOCK PUBLIC utl_SignalColumn
VAR_INPUT
	I_STS_Error:BOOL;				//Status any machine-part is in error (any organiser in error state)
	I_STS_Running:BOOL;				//Status all machine-parts are running (all organisers in Auto_K)
	I_STS_NoDischarge:BOOL;			//Status discharge (next machine) not accepting products
	I_STS_OperatorInput:BOOL;		//Status any machine-part needs operator interaction
END_VAR

VAR
	Q_H_Error AT %Q*:BOOL;			//Lamp signal error: 												RED
	Q_H_Running AT %Q*:BOOL;		//Lamp signal running:												GREEN
	Q_H_Operator AT %Q*:BOOL;		//Lamp signal operator interaction needed (refill products etc):	WHITE
END_VAR

Q_H_Error := I_STS_Error 
			OR (	I_STS_NoDischarge
					AND BknGlbl.Blink_1s);
Q_H_Running := I_STS_Running;
Q_H_Operator := I_STS_OperatorInput;

END_FUNCTION_BLOCK

// ---- _Control_Templates/cntrl_SafetyController/cntrl_SafetyController1.TcPOU
(*	TODO TEMPLATE SAFETYZONE >> change to your needs
	This is a template for a twinsafe safety project
		*Multiple groups are controlled in this example, but you can also chose to create a block per group > easier to create modules
	
	It should cover the basic needs, but you will have to adapt this as needed
	This block extends cntrl_SafetyLogic from the library
		minimal updates needed:
		-add/rename inputs and errors for es-pushbuttons/-doors/-lightbarriers/etc

	Base functionality:
		After a firstscan, the safety group is started and the error is acked. This will put the safety group in run if there are no active errors present
		In run the safety circuit can be restarted by the operator.
		
		If the group leaves run state then this is detected as an hardware error. 
		This must be reset with a dedicated reset es-stop errors button on the HMI >> PbSf_ResetSafetyErrors
		
		
	Usage:
		-DO NOT: send restart signal via the plc, this signal should be connected to a real input to twinsafe via a safe input terminal.
		-the err-ack signal is handled in the base block via HMI.STS > in the HMI it should be obvious to the user that a safety error occured and thus a safey issue is present
		-in twinsafe for groups / blockinstance you need to monitor (estop/mon/muting):
			>map state = true (so you can link via hw-terminal)
		-in twinsafe/targetsystem > set checkmark: "map crc" link to this block's crc input
			after the safety is checked by the safety-officer	

*) 

FUNCTION_BLOCK cntrl_SafetyController1 EXTENDS cntrl_SafetyLogic
VAR_INPUT
	I_HMI_Parent:ItfHMI;								//HMI of the parent block. If this block is in error, it will set the parent P_StsInError property
	I_OrgControl: ItfOrgControl;						//Organiser control bits
	
	//TODO template: remove if not needed
	I_K_EnableLsRejectMuting:BOOL;						//Signal enable muting of lightcurtain reject
	
	//TODO template: remove if not needed
	I_STS_AirPressure_OK:BOOL;							//Status airpressure ok >> needed for the safety logic to only enable safe air if pressure is valid (otherwise safety errors will occur)
END_VAR
VAR_OUTPUT
	//TODO template: add/rename zones as needed
	Q_K_ES_Zone1_OK:BOOL;								//safety circuit zone 1 ok
	Q_K_ES_Zone1_TOFOK:BOOL;							//safety circuit zone 1 delayed off ok
	Q_K_ES_Zone2_OK:BOOL;								//safety circuit zone 2 ok
END_VAR
VAR
(*Configuration*)	

(*Logged variables*)

(*Internals*)

(*Instances*)
	HMI:HMI_SafetyController1;								//All HMI related variables

(*IO*)
	//These outputs are defined in the baseblock (always used):
		//Qsf_K_RunSafety
		// Qsf_K_ResetSafetyErrors
	
	//TODO TEMPLATE
		//Add/Remove safety groups
		SFG_Hardware_Run:cntrl_safeGroup;					//Safetygroup hardware (inputs etc / plc communication)
		SFG_Zone1_Run:cntrl_safeGroup;						//Safetygroup zone 1
		SFG_Zone2_Run:cntrl_safeGroup;						//Safetygroup zone 2
		SFG_ZoneAll_Run:cntrl_safeGroup;					//Safetygroup zone All
	
		//Add/Remove safety zones
		ES_Zone1:cntrl_safeEstop;							//emergency stop zone 1
		ES_Zone2:cntrl_safeEstop;							//emergency stop zone 2
	
		//Add/remove safety devices (pushbuttons/lightscreen/etc) to create errors/statusses for the HMI
		//you can go 2 ways here
			//easy way if each door / pb-es is connected seperately (not in series) to a twinsafe terminal
				//>>use for each device a safeMon block and set in properties "map state = true" now link this output to the boikon library equivalent block
				//in this template block it is assumed this is the case
			//more work and no twinsafe-state-loggging: each pb/door is wired by an extra contact to the plc-unsafe inputs only for diagnostics / HMI-errors
				//use cntrl_InputHmiStsErr
		//everything is wired seperately to safe terminals and setting "map state = true" for the twinsafe mon blocks.
		PB_ES_MainCabinet: cntrl_safeMon;					//Pushbutton main cabinet
		DR_Front:cntrl_safeMon;								//Door infeed
		LS_Entry1:cntrl_safeMuting;							//Lightscreen entry 1

		//Add/Remove alias connections
		// this is needed if you have the boikon safety valves in the safetygroup. This will prevent activating safeair if there is no air supply (otherwise it would cause a safe-air-edm error)
		Qsf_K_EnableSafeAir AT%Q*:BOOL;						//Status airpressure is ok
END_VAR

//call baseblock functionality, handles:  resetting / starting / error detection of the safety program
SUPER^._M_StepConditions(
		//TODO TEMPLATE: request the correct key from the safety officer, otherwise you will get a safety project is not verified warning >> required by the NEN-NORMS
		I_CrcKey:= 16#1A93E370,
		//TODO TEMPLATE: adapt to nr of groups
		I_GroupsInRun:= SFG_Hardware_Run.Q_STS_OK
						AND SFG_Zone1_Run.Q_STS_OK
						AND SFG_Zone2_Run.Q_STS_OK
						AND SFG_ZoneAll_Run.Q_STS_OK, 
						//NOTE: this is 1 way of handling multiple groups.
						//the disadvantage is that if 1 groups has an issue, all groups are reset (cycled stop > reset > run)
						//if you don't want this then create extra cntrl_SafetyController(s) for group(s) that have to be independant
		IO_HMI_WRN:= HMI.WRN,		
		IO_HMI_ERR:= HMI.ERR,
		IO_HMI_STS:= HMI.STS);	
SUPER^._M_Activations(
		IO_HMI_ERR:= HMI.ERR,
		IO_HMI_STS:= HMI.STS);


//update HMI variables
_A_HMI();

//io linked to safety logic via mapped states
SFG_Hardware_Run(
	I_HMI_Parent:= HMI, 
	I_OrgControl:= I_OrgControl, 
	I_K_SimulationActive:= I_K_SimulationActive);
	
SFG_Zone1_Run(
	I_HMI_Parent:= HMI, 
	I_OrgControl:= I_OrgControl, 
	I_K_SimulationActive:= I_K_SimulationActive);
	
SFG_Zone2_Run(
	I_HMI_Parent:= HMI, 
	I_OrgControl:= I_OrgControl, 
	I_K_SimulationActive:= I_K_SimulationActive);
	
SFG_ZoneAll_Run(
	I_HMI_Parent:= HMI, 
	I_OrgControl:= I_OrgControl, 
	I_K_SimulationActive:= I_K_SimulationActive);
	
ES_Zone1(
	I_HMI_Parent:= HMI, 
	I_OrgControl:= I_OrgControl, 
	I_K_SimulationActive:= I_K_SimulationActive, 
	Q_STS_OK=> Q_K_ES_Zone1_OK, 
	Q_STS_TOF_OK=> Q_K_ES_Zone1_TOFOK);

ES_Zone2(
	I_HMI_Parent:= HMI, 
	I_OrgControl:= I_OrgControl, 
	I_K_SimulationActive:= I_K_SimulationActive, 
	Q_STS_OK=> Q_K_ES_Zone2_OK);
		
PB_ES_MainCabinet(
	I_HMI_Parent:= HMI, 
	I_OrgControl:= I_OrgControl, 
	I_K_SimulationActive:= I_K_SimulationActive);

DR_Front(
	I_HMI_Parent:= HMI, 
	I_OrgControl:= I_OrgControl, 
	I_K_SimulationActive:= I_K_SimulationActive);
	
LS_Entry1(
	I_HMI_Parent:= HMI, 
	I_OrgControl:= I_OrgControl, 
	I_K_SimulationActive:= I_K_SimulationActive,
	I_K_EnableMuting:=I_K_EnableLsRejectMuting);

	
//io linked to alias devices safety logic
	//if airpressure ok and reset pressed >> enable safe air
	//the reason behind this is to prevent EDM errors if the main air is offline and the e-system would try to enable air >> would cause edm error on sensor check
	Qsf_K_EnableSafeAir S= 	I_OrgControl.Reset_K_RE
							AND I_STS_AirPressure_OK;
	Qsf_K_EnableSafeAir R= NOT I_STS_AirPressure_OK;

ACTION _A_HMI:
//Update HMI variables (check error status + reset, check warnings)
HMI.M_Update(	I_OrgControl:= I_OrgControl,
				I_HMI_Parent:= I_HMI_Parent,
				I_ERR:= HMI.ERR,
				I_WRN:= HMI.WRN,
				I_MAN:= HMI.MAN);
				
//Warnings
				
//Errors

//Statusses
	HMI.STS.CrcCodeProject := Isf_STS_CrcSafetyProject;
END_ACTION

END_FUNCTION_BLOCK

// ---- _Control_Templates/cntrl_SafetyController/HMI_SafetyController1.TcPOU
(*	HMI variables

	This block holds all HMI variables and handles communication with the HMI
	
	2024-02 HP
		-initial
*)

{attribute 'no_explicit_call' := 'do not call this POU directly'}
FUNCTION_BLOCK HMI_SafetyController1 EXTENDS HMI_BaseBlock
//HMI variables that can be written to by the plc and HMI 
VAR_INPUT
	//Do not change these names, the HMI is hardcoded to use these exact names
	MAN:HMI_NotUsed;				//HMI manuals
	STS:HMI_STS_SafetyController1;		//HMI statusses
	WRN:HMI_WRN_SafetyController1;		//HMI warnings
	ERR:HMI_ERR_SafetyController1;		//HMI errors
END_VAR

//Hmi variables that can only be written to by the HMI and read by the plc
VAR_OUTPUT PERSISTENT
	//Do not change these names, the HMI is hardcoded to use these exact names
	//SP:HMI_SP_SafetyLogic;			//HMI setpoints
END_VAR

//this block should not be called

END_FUNCTION_BLOCK

// ---- _Scam/SCM_TemplateClean/SCM_TemplateClean.TcPOU
(*Clean SCAM template. 
	To be used as base for new projects.
	Make a copy and rename as defined in the control overview scheme
	
	Code conventions:
		Var in/out/in_out
			I_	>>block input
			Q_	>>block output
			for in+outputs:
				+K	>>Command, usually connected to potential free contacts / activation of relais.  
				+SN	>>Signal, communication with other blocks with interlocking
					+SUP	>>to/from supply (previous machinepart in the productflow)
					+DSC 	>>to/from discharge (next machinepart in the productflow)
					*A command to another block has a response with a signal with the same name but appended with _OK
						example: command= Q_SN_SUP_DeliverProduct response= I_SN_SUP_DeliverProduct_OK
				+STS	>>Status, a general status output not meant as communication with interlocking 
			
			IO_	>>block in-/output
				+HMI_ERR_[blockname] >> this struct holds all errors. !Errors should be SET, is is reset by I_OrgControl.Reset_K !In the HMI don't use errors for indicators etc
				+HMI_WRN_[blockname] >> this struct holds all warning. Warnings can be A: / S: / R:
				+HMI_STS_[blockname] >> this struct holds all statusses and possibly also buttons which are not for manual mode
				+HMI_SP_[blockname]	 >> this struct holds all setpoints. !Only read in the plc!!! Setting on plc side will not save new value in the HMI recipe!
				+HMI_MAN_[blockname] >> this struct holds all manual buttons. It is completely reset if the organiser leaves manual mode (only put buttons here, position/speed/etc can be put in statusses >>IO_STS.MAN_ABSPOS) 
				+STS	>>status
		
		Var internal
			eS		>>main state
			eE		>>exception state
			CFG_	>>configuration set by FB_Init
			HM_		>>block internal for a basetype variable
			
		Instance declarations
			Tmr_	>>TON timer
			TmrOff_	>>TOF timer
			Re		>>rising edge (R-Trig)
			Fe		>>falling edge (F-Trig)
			Cam		>>camera
			Cyl		>>cylinder (cntrl_Valve)
			Vlv		>>valve (cntrl_Valve)
			Mtr		>>Motor
			Fdr		>>Frequency drive
			Srv		>>servo
			Vcg		>>Vacuum generator
			//Inputs
			Dr		>>door
			Pb		>>pushbutton
			Pc		>>photocell
			Px		>>proximity sensor (capacitive/inductive)
			Ps		>>pressure sensor
			Rs		>>reed switch
			//Outputs
			K		>>relais
			Y		>>klep

					
			Example: Srv_LaserHeight / Cyl_TapeCutter / Tmr_CutDelay
				
			*Logged variables do not have a defined prefix yet >> try to make them logical
			if logging a position of Srv_HeightLaser then name it: Srv_HeightLaserPos
				>> now in plc lab you will find the channel below the channel where its state is logged. 
		
		Activation/Method/Properties		
			A_	>>Activation
			M_	>>Method
			P_	>>Property
			
		Conditions
			don't mix OR / AND without paranthesis (you will get bitten by the fact there is an order of precedence otherwise)
			after a paranthesis add / remove a TAB when opening / closing  
			after a condition add a ENTER
			Example:
			IF(	myBool1
				AND(	mybool2
						OR mybool3)
				AND mybool4)
			THEN
				....
			END_IF
			
		Arrays/For-loops
			define arrays with constants: 
				HM_FifoProducts: array [0..Glcn.MaxIndexFifoProducts] of ProductInfo
			if you need to loop this array then use this constant:
				FOR HM_Index:=0 TO Glcn.MaxIndexFifoProducts BY 1 
				DO
					..
				END_FOR
		
	Changes
		2019-12 HP
			-New tc3 template
		DateTime.Now() HP
			-this blocks keeps being updated with new blocks/styles/etc
		2024-02 HP
			-new hmi struct
		2025-10 HP
			-Better split of activations over actions
		
*)

FUNCTION_BLOCK SCM_TemplateClean

VAR CONSTANT
END_VAR

VAR_INPUT
	I_Organiser: ItfOrgControl;								//Organiser control bits
	//todo template>> remove if not needed
	//I_SP_GeneralShared:REFERENCE TO HMI_SP_GeneralShared; 	//General shared setpoints for multiple blocks
	
	I_K_ES_OK:BOOL;											//Signal emergency stop ok >> used for controls as extra safety to stop them no matter organiser state
	I_STS_SUP_Empty:BOOL;									//Status supply is empty >> used to detect if this block has run empty as well (sup_empty + conveyor on for x time >> this part is empty)
END_VAR

VAR_OUTPUT
	Q_STS_Empty:BOOL;								//Status this part is empty (go in energy saving / standby mode, stop conveyors etc)
END_VAR

VAR
	(*Configuration*)	

	(*Logged variables*)
	LogXaxis: utl_LoggedReal(LoggingGroup:= eLogGroups.Default , TrigAtInterval:=1 , TrigAtDeviation:=1 );
	LogYaxis: utl_LoggedReal(LoggingGroup:= eLogGroups.Default , TrigAtInterval:=1 , TrigAtDeviation:=1 );
	LogZaxis: utl_LoggedReal(LoggingGroup:= eLogGroups.Default , TrigAtInterval:=1 , TrigAtDeviation:=1 );
	
	(*Internals*)
	HMI:HMI_TemplateClean;					//All Hmi variables
	State:sTpc;								//Program state
	eE:	(U_0,U1_0,U1_1,U1_2	);				//Main state exceptions
	HM_ProgStatus:ProgStatus;				//Program general status bits	
	HM_LastTicksStateRest:ULINT;			//System ticks value last time left rest state
	HM_Empty:BOOL;							//Internal machinepart is empty
		
	(*Instances*)
	//Cyl_InfStopper:....					//Cylinder infeed stopper
	Srv_Xaxis: cntrl_Servo(
		TMR_PowerSave:=T#1M,			//time before entering powersave mode 0=disabled (if no command is given then power down after this time @ any command is reset timer) !It takes some time to awake the servo
		EnableSoftLimits:=TRUE,		//enable software limits (with button manual disable hw-limits, the parameter in the nc-task is set to 0, we need to know if it should be reenabled afterwards
		InputNrHomingSensor:=-1,			//input nr for the sensor in "axis_ref_Extended.I_DigitalInputs" -1 == disabled
		InputNrHwLimitNeg:=-1,			//input nr for the sensor in "axis_ref_Extended.I_DigitalInputs" -1 == disabled
		InputNrHwLimitPos:=-1,			//input nr for the sensor in "axis_ref_Extended.I_DigitalInputs" -1 == disabled
		JogMinusOffHomeSensor:=FALSE,	//"jog-"  when moving off homing sensor (if false then jog+ is used) in homing function
		HomingsensorIs_NC:=FALSE,		//the homing sensor is of type normally closed (note limitswitches are always normally closed)
		TmrErr_JogOffHomeSensor:=T#3S,	//time to try and jog off homing sensor t#0S = disable
		HomeTorqueSpeed:=0,						//Speed to use for homing in torque mode
		HomingMode:= eSrvHomingModes.Set,	//homing mode to use >> Default, Direct, Set, Reset, TorquePositiveDirection, TorqueNegativeDirection
		CouplingSyncPosFirst:=FALSE,			//at couple command, sync the position first to the master axis
		SPD_CouplingSyncSpeed:=0,				//speed to use when syncing position for coupling
		DST_CouplingSyncMaxDiff:=0,				//max difference allowed when sync couling >> otherwise error
		//MAKE SURE VALUE IS CORRECT (set to 0 to use nc-task configured dynamics)
		DEC_EmergencyError:=1000,			//deceleration ramp to use for emergency/error situation <= 0 means use default ramp
		//SET LOWER!!! >> jog=50, velo=250
		SPD_JOG_Max:=200,					//max allowed allowed jog speed (also used to jog of homing sensor during homing)
		SPD_AbsModVel_MaxMan:=200			//max allowed speed in manual absolute,velocity, modulo mode	
		);
		
	Srv_Yaxis: cntrl_Servo(
		TMR_PowerSave:=T#1M,			//time before entering powersave mode 0=disabled (if no command is given then power down after this time @ any command is reset timer) !It takes some time to awake the servo
		EnableSoftLimits:=TRUE,		//enable software limits (with button manual disable hw-limits, the parameter in the nc-task is set to 0, we need to know if it should be reenabled afterwards
		InputNrHomingSensor:=-1,			//input nr for the sensor in "axis_ref_Extended.I_DigitalInputs" -1 == disabled
		InputNrHwLimitNeg:=-1,			//input nr for the sensor in "axis_ref_Extended.I_DigitalInputs" -1 == disabled
		InputNrHwLimitPos:=-1,			//input nr for the sensor in "axis_ref_Extended.I_DigitalInputs" -1 == disabled
		JogMinusOffHomeSensor:=FALSE,	//"jog-"  when moving off homing sensor (if false then jog+ is used) in homing function
		HomingsensorIs_NC:=FALSE,		//the homing sensor is of type normally closed (note limitswitches are always normally closed)
		TmrErr_JogOffHomeSensor:=T#3S,	//time to try and jog off homing sensor t#0S = disable
		HomeTorqueSpeed:=0,						//Speed to use for homing in torque mode
		HomingMode:= eSrvHomingModes.Set,	//homing mode to use >> Default, Direct, Set, Reset, TorquePositiveDirection, TorqueNegativeDirection
		CouplingSyncPosFirst:=FALSE,			//at couple command, sync the position first to the master axis
		SPD_CouplingSyncSpeed:=0,				//speed to use when syncing position for coupling
		DST_CouplingSyncMaxDiff:=0,				//max difference allowed when sync couling >> otherwise error
		//MAKE SURE VALUE IS CORRECT (set to 0 to use nc-task configured dynamics)
		DEC_EmergencyError:=1000,			//deceleration ramp to use for emergency/error situation <= 0 means use default ramp
		//SET LOWER!!! >> jog=50, velo=250
		SPD_JOG_Max:=200,					//max allowed allowed jog speed (also used to jog of homing sensor during homing)
		SPD_AbsModVel_MaxMan:=200			//max allowed speed in manual absolute,velocity, modulo mode	
		);
		
	Srv_Zaxis: cntrl_Servo(
		TMR_PowerSave:=T#1M,			//time before entering powersave mode 0=disabled (if no command is given then power down after this time @ any command is reset timer) !It takes some time to awake the servo
		EnableSoftLimits:=TRUE,		//enable software limits (with button manual disable hw-limits, the parameter in the nc-task is set to 0, we need to know if it should be reenabled afterwards
		InputNrHomingSensor:=-1,			//input nr for the sensor in "axis_ref_Extended.I_DigitalInputs" -1 == disabled
		InputNrHwLimitNeg:=-1,			//input nr for the sensor in "axis_ref_Extended.I_DigitalInputs" -1 == disabled
		InputNrHwLimitPos:=-1,			//input nr for the sensor in "axis_ref_Extended.I_DigitalInputs" -1 == disabled
		JogMinusOffHomeSensor:=FALSE,	//"jog-"  when moving off homing sensor (if false then jog+ is used) in homing function
		HomingsensorIs_NC:=FALSE,		//the homing sensor is of type normally closed (note limitswitches are always normally closed)
		TmrErr_JogOffHomeSensor:=T#3S,	//time to try and jog off homing sensor t#0S = disable
		HomeTorqueSpeed:=0,						//Speed to use for homing in torque mode
		HomingMode:= eSrvHomingModes.Set,	//homing mode to use >> Default, Direct, Set, Reset, TorquePositiveDirection, TorqueNegativeDirection
		CouplingSyncPosFirst:=FALSE,			//at couple command, sync the position first to the master axis
		SPD_CouplingSyncSpeed:=0,				//speed to use when syncing position for coupling
		DST_CouplingSyncMaxDiff:=0,				//max difference allowed when sync couling >> otherwise error
		//MAKE SURE VALUE IS CORRECT (set to 0 to use nc-task configured dynamics)
		DEC_EmergencyError:=1000,			//deceleration ramp to use for emergency/error situation <= 0 means use default ramp
		//SET LOWER!!! >> jog=50, velo=250
		SPD_JOG_Max:=200,					//max allowed allowed jog speed (also used to jog of homing sensor during homing)
		SPD_AbsModVel_MaxMan:=200			//max allowed speed in manual absolute,velocity, modulo mode	
		);	
	
	(*Inputs / Outputs*)	
END_VAR

(*
	Machinepart not enabled >> note: optional remove setpoint and this code if not needed!
*)
	//If this part is not enabled >> ...
	IF (	NOT HMI.SP.MachinePartEnabled)
	THEN
		//if not disabled yet >> reset outputs + errors + warnings
		IF(	State.eS <> eTpc.Disabled)
		THEN
			//Make sure output of devices are turned off by setting state total reset and then running activations once
			State.M_Step(I_NewStep:= eTpc.Disabled);
			A_ActivationsInit();
			A_ActivationsAlways();
			
			//reset HMI variables
			utl_Any_Reset(I_Data:= HMI.ERR);
			utl_Any_Reset(I_Data:= HMI.WRN);
		END_IF

		Q_STS_Empty := I_STS_SUP_Empty;
		RETURN;
	END_IF

(*
	Update HMI variables
	Check if an error is active >> set Q_ProgStatus.Prog_Errror
*)
	HMI.M_Update(	I_OrgControl:= I_Organiser, 				//used for reset manuals/errors commands
					I_HMI_Parent := 0, 							//This is top level, no error propagation
					I_ERR:= HMI.ERR,							//The update function will check for error changes (signal to the hmi to update errors) + reset errors
					I_WRN:= HMI.WRN,							//The update function will check for warning changes (signal to the hmi to update errors)
					I_MAN:= HMI.MAN);							//The update function will reset manuals @ organiser request

(*	Simulation*)
	//if simulation active >> ..
	IF(Glbl.Sim_MyMachinePart) THEN A_Simulation();END_IF 

(*	Exceptions & step-controller*)
	A_Exceptions();

(*	State transitions*)
	//if not in exception >> execute state transitions
	IF ( 	NOT HM_ProgStatus.Prog_Exception)
	THEN 
		A_StepTransitions();
	END_IF

(*	Activations*)
	//Reset all activations controlled by states
	A_ActivationsInit();
	//Activations controlled by state
	A_ActivationsState();
	//Activations not controlled by state + instance calls
	A_ActivationsAlways();
	
(*update organiser with scam status*)
	A_UpdateOrganiserProgstatus();

ACTION A_ActivationsAlways:
(*
	State undependant activations + instance calls
*)

//Internal flags
	//Reset empty status
	IF (	NOT I_STS_SUP_Empty
			AND I_Organiser.Auto_K)
	THEN
		HM_Empty := FALSE;
	END_IF

//Warnings/Statusses	
	Q_STS_Empty := HM_Empty;
	HMI.STS.IsEmpty := HM_Empty; //can be used for a indicator (green/grey circle) on the HMI this machinepart is empty
	
	//TODO TEMPLATE
	//usually only done when connected to an external machine (customer) >> remove warning if not needed
	HMI.WRN.NotRdyRcv_Discharge := 	I_Organiser.EnableDevices_K
									AND FALSE;
	HMI.WRN.Standby := 	I_Organiser.EnableDevices_K
						AND HM_Empty;

//Timers
	//Tmr_...

//Instance calls		
	//Cyl_....
	//Srv_....	
	//etc

	Srv_Xaxis(
		I_HMI_Parent:= HMI,
		I_PTR_MasterAxis:= Srv_Xaxis.P_PointerToAxisRefExtended, 
		I_K_SimulationActive:= Glbl.Sim_MyMachinePart, 
		I_ES_OK:= I_K_ES_OK,
		I_OrgControl:= I_Organiser, 
		//..several commands.. 
		I_CPF_CoupleFactor:= 1,
		I_K_ExternalSetpoint:= FALSE);
		
	Srv_Yaxis(
		I_HMI_Parent:= HMI,
		I_PTR_MasterAxis:= Srv_Yaxis.P_PointerToAxisRefExtended, 
		I_K_SimulationActive:= Glbl.Sim_MyMachinePart, 
		I_ES_OK:= I_K_ES_OK,
		I_OrgControl:= I_Organiser, 
		//..several commands.. 
		I_CPF_CoupleFactor:= 1,
		I_K_ExternalSetpoint:= FALSE);
		
	Srv_Zaxis(
		I_HMI_Parent:= HMI,
		I_PTR_MasterAxis:= Srv_Zaxis.P_PointerToAxisRefExtended, 
		I_K_SimulationActive:= Glbl.Sim_MyMachinePart, 
		I_ES_OK:= I_K_ES_OK,
		I_OrgControl:= I_Organiser, 
		//..several commands.. 
		I_CPF_CoupleFactor:= 1,
		I_K_ExternalSetpoint:= FALSE);
		
	//Logging
	LogXaxis.V:= Srv_Xaxis.P_STS_Actposition;
	LogYaxis.V:= Srv_Yaxis.P_STS_ActPosition;
	LogZaxis.V:= Srv_Zaxis.P_STS_ActPosition;
END_ACTION

ACTION A_ActivationsInit:
(*	
	Initialisation of state dependant activations
*)

HM_ProgStatus.Prog_Rest := FALSE;
END_ACTION

ACTION A_ActivationsState:
(*
	State dependant activations
*)
CASE State.eS OF
	eTpc.TotalReset:
		//Controls
		//Internals
		//Warnings/Errors

	eTpc.Initialise:
		//Controls
		//Internals
		//Warnings/Errors

	eTpc.Rest:
		//Controls
			HM_ProgStatus.Prog_Rest := TRUE;
		//Internals
		//Warnings/Errors
		
(*  use for copy-pasting
	eTpc.:
		//Controls
		//Internals
		//Warnings/Errors
*)
END_CASE
END_ACTION

ACTION A_Exceptions:
(* State transition controller
	Handles multistep + step hold + statusses for hmi + logging*) 
		//>>must be before all method calls, since the input arguments are used
	State(I_OrgControl := I_Organiser);


(*Exceptions
	Here exeptions are handled.
	*most basic version:
		Rest U_0 := Q_ProgStatus.Prog_Exception:=false
			the main program is executed

		Rest >> Error := Q_ProgStatus.Prog_Exception:=true
		1)	@ any error >> exception state (U1_0)
			this will freeze the main program states
		2)	if the organiser is back in an automatic state and there are no errors
			it will step to U1_2 and from there to the idle state U_0
			*TODO TEMPLATE >> if needed, do actions on this transition (rarely used)
				But you could for example at a specific error force the main program to a recovery step
			
		Rest >> Totalreset := Q_ProgStatus.Prog_Exception:=true
		1)	@ organiser total reset command >> exception total reset (U1_1)
		
		2)	@ NOT organiser total reset command >> 
				>> now bits that need to be reset @ total reset are reset
				TODO Template >> add bits which needs to be reset
				>> the main program is reset to the first step (usually named: TotalReset)
				>>back to rest (U_0)

	**this described the basic version which can be used in 99% of the cases,
	you can adapt it to your needs. 
*)

CASE eE OF
	//rest
	U_0:
		//if program in error >> to error state
		IF(	HM_ProgStatus.Prog_Error
			AND NOT I_Organiser.TotalReset_K)
		THEN
			//>>
			eE := U1_0;
		//else if total reset command >> to total reset state
		ELSIF(	I_Organiser.TotalReset_K)
		THEN
			//>>
			eE := U1_1;
		END_IF

	//error
	U1_0:
		//if total reset command >> to total reset state
		IF(	I_Organiser.TotalReset_K)
		THEN
			//>>
			eE := U1_1;
			
		//else if no error active and organiser back in an automatic state
		ELSIF(	NOT HM_ProgStatus.Prog_Error
				AND I_Organiser.EnableDevices_K)
		THEN
			//>>
			eE := U1_2;
		END_IF

	//Total Reset
	U1_1:
 		//if total reset command dropped >> Reset program data and to unfreeze state
		IF(	NOT I_Organiser.TotalReset_K)
		THEN
			//Total reset main program
			State.M_Step(
				I_NewStep:= eTpc.TotalReset,
				I_StepCanBeHeld:= TRUE);
			
			//disable multistepping for 1 round
			{warning disable C0139}
			State.P_IsMultiStepRequired;
			
			//>>
			eE := U_0;
		END_IF
		
	//Unfreeze
	U1_2:
		//>>
		eE := U_0;

	ELSE
		eE := U_0;
END_CASE
//Detection program in exception
HM_ProgStatus.Prog_Exception := (eE > U_0);
END_ACTION

ACTION A_Simulation:
(*
	Code that only needs to be executed if simulation is active (this action is only called if sim is active)

	Notes:	
	-Cntrl_Servo/motor/valve already simulate their state correctly themselves, cntrl_StateSensor must be told which state to simulate >> example below
		Of course you could also add timers / other conditions (servo pos?!) for states
	
*)

//Initialise activations, which are controlled by the simulation steps
//fbPC_Example.I_SimulateState := eSensorState.Undetected;


(*Step activations*)
CASE State.eS OF
	eTpc.TotalReset:
	;

	eTpc.Rest:
		//Example simulate sensor ON immediatly
			//fbPC_Example.I_SimulateState := eSensorState.Detected;
		
		//Example simulate sensor ON in a step after a delay
			//IF(Step.P_StepTime > T#33MS) THEN fbPC_Example.I_SimulateState := eSensorState.Detected; END_IF
		
END_CASE
END_ACTION

ACTION A_StepTransitions:
(*In this section all state transitions are made

	-no activations are done here (do this in A_Activations)
	-The transition to a new step is the ideal location to do rising edge settings
		IF(myCondition) THEN
			HM_CNT_Example := HM_CNT_EXAMPLE + 1; //example to count something
			fbSrv_Example.I_POS_Auto_Absolute := myNewPosition + someCalculated offset; //example to calculate endpoint for a servo
			//Note: you could set the servo speed here as well, but then you can't change the speed anymore during the movement
				probably (dependant on your situation) better to do it in activations.
			//>>
			step to next step
		END_IF

*)

(*Main program steps*)

//if stepping not locked, by steplock mode >> can be toggled in HMI to lock certain steps for commissioning/debugging
IF( NOT State.Q_K_LockSteps)
THEN
//Repeat until conditions to step to next state are false OR looped already twice (normally programs don't loop multiple times!)
REPEAT 
	CASE State.eS OF
		eTpc.Disabled,
		eTpc.TotalReset:
			//if initialise command from the organiser																>>Initialise
				IF ( I_Organiser.Init_K)
				THEN
					//>>
					State.M_Step(
						I_NewStep:= eTpc.Initialise,
						//Optional: argument to log extra info for this step transition
						I_NewStepLogInfo:= CONCAT('TotalReset:', SYSTEMTIME_TO_STRING(BknGlbl.LocalSystemTime)),
						//>>@ true & HMI-stepmode is activated, then the next state will be locked until you press the button release step on the HMI (used for debugging / commissioning
						//!Do not enable for states in which things are cooking: (heater enabled / motor running / etc) or at least consider carefully potential dangers.
						I_StepCanBeHeld:= TRUE,
						//Optional: >> the repeat around this CASE-statement will NOT execute, the next step will take at least 1 cycle == activations for that step are executed 	
						I_BlockMultiStep:=TRUE); 
				END_IF

		eTpc.Initialise:
			//if components initialised																				>>Rest
				IF( FALSE) 
				THEN
					//>>
					State.M_Step(
						I_NewStep:= eTpc.Rest,
						I_StepCanBeHeld:= TRUE);
				END_IF

		eTpc.Rest:
			//if machine started and start condition																>>Rest
				IF( I_Organiser.Auto_K
					AND FALSE)
				THEN
					//>>
					State.M_Step(
						I_NewStep:= eTpc.Rest,
						//just an example what you can do (add state info for logging purposes), this argument is optional
						I_NewStepLogInfo:= Concat('Last cycle time(s):', TO_STRING(TO_REAL(BknGlbl.SystemTimeInTicks - HM_LastTicksStateRest)/10000000)),
						I_StepCanBeHeld:= FALSE);
					HM_LastTicksStateRest := BknGlbl.SystemTimeInTicks;
				END_IF

		(*  use for copy-pasting
				Keep tab-structure > try fold icon on comment lines for step reasons ;)
			
			eTpc.:
				//if [ReasonForStep]																				>>[TargetState]
					IF()
					THEN
						//>>
						State.M_Step(
							I_NewStep:= eTpc.,
							I_StepCanBeHeld:= TRUE);
				//else if [ReasonForStep]																			>>[TargetState]
					ELSEIF
					THEN
						
					END_IF
		*)

	//unkown state, should never happen. Best to not do an autorecovery, just let it hang			
	ELSE
		utl_SystemMessageWithLogging(I_Message:='prog error step missing');
	END_CASE 

//until flag to multistep is false 
UNTIL(NOT State.P_IsMultiStepRequired)
END_REPEAT
END_IF
END_ACTION

ACTION A_UpdateOrganiserProgstatus:
//machinepart in exception > done in A_Exceptions
//HM_ProgStatus.Prog_Exception

//machinepart in rest state > done in A_ActivationsState
//HM_ProgStatus.Prog_Rest

HM_ProgStatus.Prog_Error :=	//emergencystop not ok
							NOT I_K_ES_OK
							//error active in this block or one of the local children (cntrl_xxxx for example)
							OR HMI.P_STS_InError;

//production stopped by external factor >> for OEE performance tracking / lamp signal column 
HM_ProgStatus.Prog_ExternallyBlocked := FALSE; //TODO TEMPLATE: Activate if needed, example: NOT SN_DscReadyToReceive;

//machinepart needs attention >> for lamp signal column
HM_ProgStatus.Prog_Attention := FALSE; //TODO TEMPLATE: Activate if needed, example: PC_PlanoBufferLowLevel.Q_DetectedDebounced;

//call organiser update method
I_Organiser.M_UpdateProgStatus(HM_ProgStatus);
END_ACTION

END_FUNCTION_BLOCK

// ---- _Scam/SCM_TemplateClean/EnumsAndState/sTpc.TcPOU
(*	SCAM-State
	Lifts project unique variables to the project while keeping library functionality

	BaseBlock
		This blocks handles stuff that needs to be done @ state transitions
			-logging
			-multistepping
			-steplocking


	Usage:
		Adaptions needed to this block
		-Copy template
		-Redefine variable "eS" to your state enum
			*reasoning for var_input >> an input can be read/written to in the outside world as well as here
		
		Already done if you have copied the template
		-Finish abstract properties


	Usage in the scam:
		-This block needs to be called once before the state transitions
		-in the scam step-transitions, call the method M_Step(....) to jump to your requested state
			-in arguments define if the step can be held / log extra info
*)

FUNCTION_BLOCK sTpc EXTENDS utl_ScmState
VAR_INPUT
	eS:eTpc;  //enum holding your project unique scam-state
END_VAR

SUPER^(I_OrgControl := I_OrgControl);

//This property is used by the base block to manipulate eS since it doesn't know the enum type
PROPERTY P_StateAsInt : INT
GET
P_StateAsInt := eS;
END_GET
SET
VAR
	pInt:pointer to int;
END_VAR
//I really want to keep attribute strict for the enum definition (to prevent enum mixing which I've seen happen) but with strict you're not allowed to assign an int which must be done here!
//so let's go evil mode... 
pInt := ADR(eS);
pInt^ := P_StateAsInt;
END_SET
END_PROPERTY

//This property is used by the base block to manipulate eS since it doesn't know the enum type
PROPERTY P_StateAsString : STRING(40)
GET
P_StateAsString := TO_STRING(eS);
END_GET
END_PROPERTY

END_FUNCTION_BLOCK

// ---- DevelopmentPlayground/MurrModLight60/cntrl_MurrModLight60.TcPOU
(*


	Usage:
		In the hw-manager @io-link card >
			-auto scan for the device
			-right click the device and select process data
			-in this tab, select 'stack mode' and press activate
			-now the output image is updated and only now start linking
		Link the array of bytes while checkmark continuos is set to all outputs in 1 go
		
 
*)


FUNCTION_BLOCK cntrl_MurrModLight60
VAR_INPUT
	I_K_Error:BOOL;			//emergency stop / error active
	I_K_Alert:BOOL;			//operator assistance needed (product running out etc)
	I_K_Running:BOOL;		//machine running
END_VAR
VAR_OUTPUT
END_VAR
VAR
	CFG_NrOfStacks:BYTE;
	Q_: MurrModLight60_IO; //link to hw murr outputs
END_VAR

//the uglyness... reason type "bit3" is only an hardware thing...
Q_.Control.StacksBit0 := CFG_NrOfStacks.0;
Q_.Control.StacksBit1 := CFG_NrOfStacks.1;
Q_.Control.StacksBit2 := CFG_NrOfStacks.2;

//if error active
IF(I_K_Error)
THEN
	//set color
	Q_.Control.Stack3 := eMurrModLight60Colors.COLOR_RED;
ELSE
	Q_.Control.Stack3 := 0;
END_IF

//if alert active
IF(I_K_Alert)
THEN
	//set color
	Q_.Control.Stack2 := eMurrModLight60Colors.COLOR_YELLOW 
						+ eMurrModLight60Colors.PAT_GRADBLINK;
ELSE
	Q_.Control.Stack2 := 0;
END_IF

//if running
IF(I_K_Running)
THEN
	//set color
	Q_.Control.Stack1 := eMurrModLight60Colors.COLOR_GREEN;
ELSE
	Q_.Control.Stack1 := 0;
END_IF

//FB_Init is always available implicitly and it is used primarily for initialization.
//The return value is not evaluated. For a specific influence, you can also declare the
//methods explicitly and provide additional code there with the standard initialization
//code. You can evaluate the return value.
METHOD FB_Init: BOOL
VAR_INPUT
    bInitRetains: BOOL; // TRUE: the retain variables are initialized (reset warm / reset cold)
    bInCopyCode: BOOL;  // TRUE: the instance will be copied to the copy code afterward (online change)

	NrOfStacks:byte;	//number of stacks to use (the one I tested with had a max of 3, but you can decrease)   
END_VAR
CFG_NrOfStacks := NrOfStacks;
END_METHOD

END_FUNCTION_BLOCK

// ---- CHECKBOUNDS.TcPOU
(*	Function that checks and limits if an array is adressed outside of its boundaries
Usage:
	-add this function to the project, it is now called automagicly by twincat everytime an array operation is performed
	
Notes:
	-This function does increase the cpu load, it is recommended by beckhoff to only have it activated for testing
	 >the function can be left in the project, just set "exclude from build" in the properties to true

		-a GLBL status bit is set and the out of bounds index is stored

Changes:
	2020-01-28 HP
		-New tc3 template
	2023-02 HP
		-new systemmessage logging
*)
{warning 'TODO Template: CHECKBOUNDS is active, this causes increased processor load. Exclude block from build when possible'}
FUNCTION CHECKBOUNDS : DINT
VAR_INPUT
        index, lower, upper : DINT;
END_VAR

//if index lower than array memory >> set to lowest possible
IF index<lower THEN
	//Variables are set (never reset unless manual/power cycle)
	.Glbl.OutOfBounds := TRUE;
	.Glbl.OutOfBoundsIndex := index;

	//set the index to lowest
	CHECKBOUNDS := lower;
	
	//log system message
	utl_SystemMessageWithLogging(I_Message:=CONCAT('Checkbounds lower violation detected:',TO_STRING(index)));
	
//if index higher than array memory >> set to highest possible
ELSIF index>upper THEN
	//Variables are set (never reset unless manual/power cycle)
	.Glbl.OutOfBounds:=TRUE;
	.Glbl.OutOfBoundsIndex := index;
	
	//set the index to lowest
	CHECKBOUNDS := upper;

	//log system message
	utl_SystemMessageWithLogging(I_Message:=CONCAT('Checkbounds upper violation detected:',TO_STRING(index)));

//else index is within array memory
ELSE
	CHECKBOUNDS := index;
END_IF

END_FUNCTION

// ---- DevelopmentPlayground/ObjectOrientedExamples/OopExmplBase.TcPOU
(*	This block is defined with the "ABSTRACT" keyword. This means it can not be used  directly, it can only be used to be expanded upon
		>>create a new function which "EXTENDS" this block and add extra stuff as needed
*)
FUNCTION_BLOCK ABSTRACT OopExmplBase
VAR_INPUT
	I_Base:BOOL;
	//object as input, with known interface
	I_ObjectWithGivenInterface:IOopExmpl; //note: this will crash the plc if nothing is connected at the line where this input is used
END_VAR
VAR_OUTPUT
	Q_Base:BOOL;
END_VAR
VAR_IN_OUT

END_VAR
VAR
	HM_Base:BOOL;
END_VAR

//we know the object at this input has the given interface, so it must have the interface method and we can use this
HM_Base := I_ObjectWithGivenInterface.MustHaveMethod(I:=I_Base);
Q_Base := HM_Base;

END_FUNCTION_BLOCK

// ---- DevelopmentPlayground/ObjectOrientedExamples/OopExmplExtension.TcPOU
(*	Extending the base block

*)
FUNCTION_BLOCK OopExmplExtension EXTENDS OopExmplBase
VAR_INPUT
	I_Extension:BOOL;
END_VAR
VAR_OUTPUT
	Q_Extension:BOOL;
END_VAR
VAR
	HM_Extension:BOOL;
END_VAR

//call baseblock functionality
SUPER^();

//extra code added by extension
HM_Extension := HM_Base AND I_Extension;
Q_Extension := HM_Extension;

END_FUNCTION_BLOCK

// ---- DevelopmentPlayground/ObjectOrientedExamples/OopExmplMain.TcPOU
(*example using the extended block with a random block that has a known interface to show how to use interfaces
*)
PROGRAM OopExmplMain
VAR
	//this block expanded the baseblock. The baseblock has an input of type interface "IOopExmpl"
	fbOopExmplExtension: OopExmplExtension;
	
	//this block implemented the interface "IOopExmpl"
	fbOopObjWithInterface: OopExmplRandomObjectWithInterface;
END_VAR

fbOopExmplExtension(
	I_Base:= , 
	Q_Base=> ,
	I_ObjectWithGivenInterface:=fbOopObjWithInterface, //note>>plc will crash if nothing is entered here (due to invalid program pointer)
	I_Extension:= , 
	Q_Extension=> );

END_PROGRAM

// ---- DevelopmentPlayground/ObjectOrientedExamples/OopExmplRandomObjectWithInterface.TcPOU
(*This block implements interface "IOopExmpl" 
	>>this means is must have the methods described in the interface

*)
FUNCTION_BLOCK OopExmplRandomObjectWithInterface IMPLEMENTS IOopExmpl
VAR
	HM_b1:BOOL; //not used for example
END_VAR

//code we are not using in the interface example
HM_b1:=TRUE;
//...
//...
//...
//...
//...

//Method the object must implement because of the interface
METHOD MustHaveMethod : BOOL
VAR_INPUT
	I:BOOL;
END_VAR
MustHaveMethod := I;
END_METHOD

END_FUNCTION_BLOCK

// ---- DevelopmentPlayground/UnitTesting/BreakLogging.TcPOU
{attribute 'no-analysis'}
FUNCTION BreakLogging : bool
VAR
	//this is bad, since var inside a function is a temp variable!
	TestLog:utl_LoggedBool(LoggingGroup:= eLogGroups.Default);
	
	//out of curiousity
	testVarInfo: __SYSTEM.VAR_INFO;
	testIoVarInfo: __SYSTEM.VAR_INFO;
END_VAR

//send message to twincat editor error list
ADSLOGSTR(
	msgCtrlMask := ADSLOG_MSGTYPE_ERROR, 
	msgFmtStr   := 'Unittesting: next error should be loggedchannel invalid path: ', 
	strArg      := '');
	
//does not work
Testlog.B := TRUE;
Testlog.B := FALSE;

//this would work (feeding an external logged channel by IO!
//IO_MyLoggedVariable.B := BknGlbl.Blink_1s;

//of course using a loggedchannel declared in a global var will work as well!
//Glbl.MyLoggedChannel.B := BknGlbl.Blink_1sec;

END_FUNCTION

// ---- _Control_Templates/cntrl_RbtFanuc/cntrl_RbtFanucUnloadingRobot.TcPOU
FUNCTION_BLOCK cntrl_RbtFanucUnloadingRobot EXTENDS cntrl_RbtFanuc
VAR_INPUT
	I_HMI_Parent:ItfHMI;		//HMI of the parent block. If this block is in error, it will set the parent P_StsInError property
	I_K_ProgramSelect:BOOL;		//Command select given program nr using the PNS-select-method
	I_K_DropBasket:BOOL;		//Command to drop basket
	I_SP_ProgramNr: BYTE;		//program nr to select
END_VAR
VAR_OUTPUT
	Q_K_ProgramSelect_OK:BOOL;	//Command select given progran nr succeeded
	Q_K_DropBasket_OK:BOOL;		//Command executed
END_VAR

VAR
	(*Configuration*)	

	(*Logged variables*)
	RbtError: utl_LoggedUInt(LoggingGroup:= eLogGroups.Cntrl_states, TrigAtInterval:= 0, TrigAtDeviation:= 0);
	RbtState: utl_LoggedUInt(LoggingGroup:= eLogGroups.Cntrl_states, TrigAtInterval:= 0, TrigAtDeviation:= 0);
	
	(*Internals*)
	TmrPayloadConfirm:TON;
	
	(*Instances*)
	HMI:HMI_RbtFanucUnloading;										//All HMI related variables
	PX_BasketLeft_X:cntrl_Sensor(Options:= eSensorConfig.InputNo );
	PX_BasketRight_X:cntrl_Sensor(Options:= eSensorConfig.InputNO );
	PC_ScanningLeft_Z:cntrl_Sensor(Options:= eSensorConfig.InputNO );
	PC_ScanningRight_Z:cntrl_Sensor(Options:= eSensorConfig.InputNO );

	Cyl_Gripper:cntrl_Valve(Options:= eValveConfig.Default + eValveConfig.HoldState);
	Cyl_Hook:cntrl_Valve(Options:= eValveConfig.None + eValveConfig.HoldState);

	(*Inputs / Outputs*)
	I_DataIn: RbtFanucUnloading_DataIn;
	Q_DataOut: RbtFanucUnloading_DataOut;
END_VAR

//call baseblock > handles base functionality like resettings / starting / selecting program
//note: the baseblock doesn't know about your custom HMI bits, but since the custom HMI bits are extended, you can supply them and the compiler will pass only the base bits
SUPER^.M_SuperCall(
	IHMI:= HMI,
	IO_StatusWord:= I_DataIn.Vars._UO,
	IO_ControlWord:= Q_DataOut.Vars._UI,
	IO_HMI_WRN:= HMI.WRN, 
	IO_HMI_ERR:= HMI.ERR, 
	IO_HMI_STS:= HMI.STS);
	
//Update HMI variables
_A_HMI();

//Simulation
IF(I_K_SimulationActive) THEN _Simulation(); END_IF

//Activations output etc
_A_Activations();

ACTION _A_Activations:

//logging
RbtError.V := I_DataIn.Vars._GO.ErrorNr;
RbtState.V := I_DataIn.Vars._GO.State;

//implementation example of how to select a program. 
//* you can also use the method from the baseblock directly in your parentblock step conditions and remove these inputs
IF( I_K_ProgramSelect
	//in the totalreset method also a program is selected, give that priority. This situation should not happen because above command should be low @total_reset but i'm a monkey
	AND_THEN eS <> eRbtFanuc.TotalReset)
THEN
	Q_K_ProgramSelect_OK := M_PNS_SelectProgram(I_SP_ProgramNr);
ELSE
	Q_K_ProgramSelect_OK:=FALSE;
END_IF

//auto confirm ready to drop (normally linked to scam, here testing real robot which is now talking to itself)
Q_DataOut.Vars._DI.SN_RequestDumpOk := I_DataIn.Vars._DO.SN_RequestDump;
Q_DataOut.Vars._DI.SN_InitLeft R= I_DataIn.Vars._DO.SN_InitLeftOk;
Q_DataOut.Vars._DI.SN_InitRight R= I_DataIn.Vars._DO.SN_InitRightOk;

//Example command from scam/response linking
Q_DataOut.Vars._DI.K_DropBasket := I_K_DropBasket;
Q_K_DropBasket_OK := I_DataIn.Vars._DO.K_DropBasket_OK;

Cyl_Gripper(
	I_HMI_Parent:= 0, 
	I_OrgControl:= I_OrgControl, 
	I_K_SimulationActive:= Glbl.SimEnable, 
	I_ES_OK:= TRUE, 
	I_K_DisableErrorDetection:= TRUE, 
	I_K_AutoIn:= I_DataIn.Vars._DO.SN_CylIn, 
	I_K_AutoOut:= I_DataIn.Vars._DO.SN_CylOut, 
	Q_STS_In=> , 
	Q_STS_Out=> );

//for now a slave as well to support left cylinder
Cyl_Hook(
	I_HMI_Parent:= 0, 
	I_OrgControl:= I_OrgControl, 
	I_K_SimulationActive:= Glbl.SimEnable, 
	I_ES_OK:= TRUE, 
	I_K_DisableErrorDetection:= TRUE, 
	I_K_AutoIn:= Cyl_Gripper.I_K_AutoIn, 
	I_K_AutoOut:= Cyl_Gripper.I_K_AutoOut, 
	Q_STS_In=> , 
	Q_STS_Out=> );

//Cylinder communication to robot >> if command in/out and status cylinder matches then respons command OK
Q_DataOut.Vars._DI.SN_CylInOk := 	I_DataIn.Vars._DO.SN_CylIn
								AND Cyl_Gripper.Q_STS_In
								AND Cyl_Hook.Q_STS_In;
								
Q_DataOut.Vars._DI.SN_CylOutOk := I_DataIn.Vars._DO.SN_CylOut
								AND Cyl_Gripper.Q_STS_Out; 


PC_ScanningLeft_Z(
	I_HMI_Parent:= 0, 
	I_OrgControl:= I_OrgControl, 
	I_K_SimulationActive:= Glbl.SimEnable, 
	I_SimulateState:= , 
	I_ErrNotState:= , 
	Q_DetectedDirect=> , 
	Q_DetectedDebounced=> Q_DataOut.Vars._DI.PC_Left_Z , 
	Q_DetectedDebounced_RE=> , 
	Q_DetectedDebounced_FE=> );
	
PC_ScanningRight_Z(
	I_HMI_Parent:= 0, 
	I_OrgControl:= I_OrgControl, 
	I_K_SimulationActive:= Glbl.SimEnable, 
	I_SimulateState:= , 
	I_ErrNotState:= , 
	Q_DetectedDirect=> , 
	Q_DetectedDebounced=> Q_DataOut.Vars._DI.PC_Right_Z , 
	Q_DetectedDebounced_RE=> , 
	Q_DetectedDebounced_FE=> );
	
PX_BasketLeft_X(
	I_HMI_Parent:= 0, 
	I_OrgControl:= I_OrgControl, 
	I_K_SimulationActive:= Glbl.SimEnable, 
	I_SimulateState:= , 
	I_ErrNotState:= , 
	Q_DetectedDirect=> , 
	Q_DetectedDebounced=> Q_DataOut.Vars._DI.PX_Left_X , 
	Q_DetectedDebounced_RE=> , 
	Q_DetectedDebounced_FE=> );
	
PX_BasketRight_X(
	I_HMI_Parent:= 0, 
	I_OrgControl:= I_OrgControl, 
	I_K_SimulationActive:= Glbl.SimEnable, 
	I_SimulateState:= , 
	I_ErrNotState:= , 
	Q_DetectedDirect=> , 
	Q_DetectedDebounced=> Q_DataOut.Vars._DI.PX_Right_X , 
	Q_DetectedDebounced_RE=> , 
	Q_DetectedDebounced_FE=> );
END_ACTION

ACTION _A_HMI:
//Update HMI variables (check error status + reset, check warnings)
HMI.M_Update(	I_OrgControl:= I_OrgControl,
				I_HMI_Parent:= I_HMI_Parent,
				I_ERR:= HMI.ERR,
				I_WRN:= HMI.WRN,
				I_MAN:= HMI.MAN);
END_ACTION

ACTION _Simulation:
//NOTE: The baseblock already resets all bits in the statusword before setting simulated bits.
//>>not doing anything (yet) with those bits here

//I_K_ProgSelect should already be simulated by the baseblock since that is default functionality
//Only custom functionality needs to be simulated here

I_DataIn.Vars._DO.K_DropBasket_OK := I_K_DropBasket;
END_ACTION

(*	Actions to be done @ Total_Reset 
	The baseblock will call this method until it returns true in state Total_Reset
	
	*if nothing special needs to be done, just return true
*)
METHOD PUBLIC M_TotalResetProcedure : BOOL
//The coloborative robot needs a signal to confirm the payload before it does anything after a power cycle. 
//You can connect it (DCS-config) to an input like is done here
TmrPayloadConfirm(IN:= TRUE, PT:= T#1.5S);
Q_DataOut.Vars._DI.SN_PayloadConfirm := TRUE;

//if done > reset vars, signal baseblock total_reset done by returning true so it can continue
IF(	TmrPayloadConfirm.Q
	//select program PNS0001 on the controller (method returns true at success)
	AND M_PNS_SelectProgram(PNS_Nr:=1))
THEN
	//reset timer + signal 
	TmrPayloadConfirm(IN:= FALSE);
	Q_DataOut.Vars._DI.SN_PayloadConfirm := FALSE;
	//signal base totale reset = done
	M_TotalResetProcedure := TRUE;
//else not done, keep baseblock in total reset state
ELSE
	M_TotalResetProcedure := FALSE;
END_IF
END_METHOD

PROPERTY PROTECTED P_ControlWord : REFERENCE TO RbtFanuc_ControlWord
GET
P_ControlWord ref= Q_DataOut.Vars._UI;
END_GET
END_PROPERTY

PROPERTY PROTECTED P_StatusWord : REFERENCE TO RbtFanuc_StatusWord
GET
P_StatusWord ref= I_DataIn.Vars._UO;
END_GET
END_PROPERTY

END_FUNCTION_BLOCK

// ---- _Control_Templates/cntrl_RbtFanuc/HMI/HMI_RbtFanucUnloading.TcPOU
(*	HMI variables

	This block holds all HMI variables and handles communication with the HMI
	
	2024-02 HP
		-initial
*)

{attribute 'no_explicit_call' := 'do not call this POU directly'}
{attribute 'analysis' := '-33'} //unused variables
FUNCTION_BLOCK HMI_RbtFanucUnloading EXTENDS HMI_BaseBlock
//HMI variables that can be written to by the plc and HMI 
VAR_INPUT
	//Do not change these names, the HMI is hardcoded to use these exact names
	MAN:HMI_MAN_RbtFanucUnloading;			//HMI manuals
	STS:HMI_STS_RbtFanucUnloading;			//HMI statusses
	WRN:HMI_WRN_RbtFanucUnloading;			//HMI warnings
	ERR:HMI_ERR_RbtFanucUnloading;			//HMI errors
END_VAR

//Hmi variables that can only be written to by the HMI and read by the plc
VAR_OUTPUT PERSISTENT
	//Do not change these names, the HMI is hardcoded to use these exact names
	SP:HMI_SP_RbtFanucUnloading;			//HMI setpoints
END_VAR

//this block should not be called

END_FUNCTION_BLOCK

// ---- _Scam/SCM_TemplateMachinePart/EnumsAndState/sTmp.TcPOU
(*	SCAM-State
	Lifts project unique variables to the project while keeping library functionality

	BaseBlock
		This blocks handles stuff that needs to be done @ state transitions
			-logging
			-multistepping
			-steplocking


	Usage:
		Adaptions needed to this block
		-Copy template
		-Redefine variable "eS" to your state enum
			*reasoning for var_input >> an input can be read/written to in the outside world as well as here
		
		Already done if you have copied the template
		-Finish abstract properties


	Usage in the scam:
		-This block needs to be called once before the state transitions
		-in the scam step-transitions, call the method M_Step(....) to jump to your requested state
			-in arguments define if the step can be held / log extra info
*)

FUNCTION_BLOCK sTmp EXTENDS utl_ScmState
VAR_INPUT
	eS:eTMP;  //enum holding your project unique scam-state
END_VAR

SUPER^(I_OrgControl := I_OrgControl);

//This property is used by the base block to manipulate eS since it doesn't know the enum type
PROPERTY P_StateAsInt : INT
GET
P_StateAsInt := eS;
END_GET
SET
VAR
	pInt:pointer to int;
END_VAR
//I really want to keep attribute strict for the enum definition (to prevent enum mixing which I've seen happen) but with strict you're not allowed to assign an int which must be done here!
//so let's go evil mode... 
pInt := ADR(eS);
pInt^ := P_StateAsInt;
END_SET
END_PROPERTY

//This property is used by the base block to manipulate eS since it doesn't know the enum type
PROPERTY P_StateAsString : STRING(40)
GET
P_StateAsString := TO_STRING(eS);
END_GET
END_PROPERTY

END_FUNCTION_BLOCK

// ---- _Scam/SCM_TemplateMachinePart/HMI/HMI_TemplateMachinePart.TcPOU
(*	HMI variables

	This block holds all HMI variables and handles communication with the HMI
	
	2024-02 HP
		-initial
*)
{attribute 'no_explicit_call' := 'do not call this POU directly'}
FUNCTION_BLOCK HMI_TemplateMachinePart EXTENDS HMI_BaseBlock

//HMI variables that can be written to by the plc and HMI 
VAR_INPUT
	//Do not change these names, the HMI is hardcoded to use these exact names
	MAN:HMI_MAN_TemplateMachinePart;			//HMI manuals
	STS:HMI_STS_TemplateMachinePart;			//HMI statusses
	WRN:HMI_WRN_TemplateMachinePart;			//HMI warnings
	ERR:HMI_ERR_TemplateMachinePart;			//HMI errors
END_VAR

//Hmi variables that can only be written to by the HMI and read by the plc
VAR_OUTPUT PERSISTENT
	//Do not change these names, the HMI is hardcoded to use these exact names
	SP:HMI_SP_TemplateMachinePart;				//HMI setpoints
END_VAR

//this block should not be called

END_FUNCTION_BLOCK

// ---- _Scam/SCM_TemplateMachinePart/SCM_TemplateMachinePart.TcPOU
(*Template step program
	
	Standard template with examples and lots of explanations >> use scm_TemplateClean as base for a new project
	This doubles as a test of all cntrl_blocks of the library (these are also used on the HMI_Template.Page_Test)
	
	
	Code conventions:
		Var in/out/in_out
			I_	>>block input
			Q_	>>block output
			for in+outputs:
				+K	>>Command, usually connected to potential free contacts / activation of relais.  
				+SN	>>Signal, communication with other blocks with interlocking
					+SUP	>>to/from supply (previous machinepart in the productflow)
					+DSC 	>>to/from discharge (next machinepart in the productflow)
					*A command to another block has a response with a signal with the same name but appended with _OK
						example: command= Q_SN_SUP_DeliverProduct response= I_SN_SUP_DeliverProduct_OK
				+STS	>>Status, a general status output not meant as communication with interlocking 
			
			IO_	>>block in-/output
				+HMI_ERR_[blockname] >> this struct holds all errors. !Errors should be SET, is is reset by I_OrgControl.Reset_K !In the HMI don't use errors for indicators etc
				+HMI_WRN_[blockname] >> this struct holds all warning. Warnings can be A: / S: / R:
				+HMI_STS_[blockname] >> this struct holds all statusses and possibly also buttons which are not for manual mode
				+HMI_SP_[blockname]	 >> this struct holds all setpoints. !Only read in the plc!!! Setting on plc side will not save new value in the HMI recipe!
				+HMI_MAN_[blockname] >> this struct holds all manual buttons. It is completely reset if the organiser leaves manual mode (only put buttons here, position/speed/etc can be put in statusses >>IO_STS.MAN_ABSPOS) 
				+STS	>>status
		
		Var internal
			eS		>>main state
			eE		>>exception state
			CFG_	>>configuration set by FB_Init
			HM_		>>block internal for a basetype variable
			
		Instance declarations
			Tmr_	>>TON timer
			TmrOff_	>>TOF timer
			Re		>>rising edge (R-Trig)
			Fe		>>falling edge (F-Trig)
			Cam		>>camera
			Cyl		>>cylinder (cntrl_Valve)
			Vlv		>>valve (cntrl_Valve)
			Mtr		>>Motor
			Fdr		>>Frequency drive
			Srv		>>servo
			Vcg		>>Vacuum generator
			//Inputs
			Dr		>>door
			Pb		>>pushbutton
			Pc		>>photocell
			Px		>>proximity sensor (capacitive/inductive)
			Ps		>>pressure sensor
			Rs		>>reed switch
			//Outputs
			K		>>relais
			Y		>>klep
					
			Example: Srv_LaserHeight / Cyl_TapeCutter / Tmr_CutDelay
				
			*Logged variables do not have a defined prefix yet >> try to make them logical
			if logging a position of Srv_HeightLaser then name it: Srv_HeightLaserPos
				>> now in plc lab you will find the channel below the channel where its state is logged.
		
		Activation/Method/Properties		
			A_	>>Activation
			M_	>>Method
			P_	>>Property
			
		Conditions
			don't mix OR / AND without paranthesis (you will get bitten by the fact there is an order of precedence otherwise)
			after a paranthesis add / remove a TAB when opening / closing  
			after a condition add a ENTER
			Example:
			IF(	myBool1
				AND(	mybool2
						OR mybool3)
				AND mybool4)
			THEN
				....
			END_IF
			
		Arrays/For-loops
			define arrays with constants: 
				HM_FifoProducts: array [0..Glcn.MaxIndexFifoProducts] of ProductInfo
			if you need to loop this array then use this constant:
				FOR HM_Index:=0 TO Glcn.MaxIndexFifoProducts BY 1 
				DO
					..
				END_FOR
		
	Changes
		2019-12 HP
			-New tc3 template
		2024-02 HP
			-new hmi struct
		DateTime.Now() HP
			-this blocks keeps being updated with new blocks/styles/etc
*)

FUNCTION_BLOCK SCM_TemplateMachinePart
VAR_INPUT
	I_Organiser: ItfOrgControl;								//Organiser control bits
	I_SP_GeneralShared:REFERENCE TO HMI_SP_GeneralShared; 	//General shared setpoints for multiple blocks
		
	I_K_ES_OK:BOOL;									//Signal emergency stop ok >> used for controls as extra safety to stop them no matter organiser state
	I_SN_SUP_Request_OK:BOOL;						//Signal supply is running AND delivering products
	I_STS_SUP_Empty:BOOL;							//Status supply is empty (used FOR energy save mode)
END_VAR

VAR_OUTPUT
	Q_SN_SUP_Request:BOOL;							//Signal supply requesting products
	Q_STS_RefillPlanos:BOOL;						//Status plano buffer needs refill 
	Q_STS_Empty:BOOL;								//this part is empty (go in energy saving / standby mode, stop conveyors etc)
END_VAR

VAR
(*Configuration*)

(*Logged variables*)
	PC_Example_Count: utl_LoggedDint(LoggingGroup:= eLogGroupsProject.Template, TrigAtInterval:= 0, TrigAtDeviation:=0 ); 	//Logged counter: example how we can count the debounced falling edges of a photocell

	//Logged servo velo example
	Srv_Example_Velo: utl_LoggedReal(
		LoggingGroup:= 	eLogGroupsProject.Template, 	//only log when this bit is set ( MAIN.visualisation ) 
						TrigAtInterval:= 10, 			//log every 10 plc cycles
						TrigAtDeviation:=1);			//Log if pos change >= 1
(*Internals*)
	State: sTmp; 											//Main state program
	eE:	(U_0,U1_0,U1_1,U1_2	);							//Main state exceptions
	HM_ProgStatus:ProgStatus;							//Program general status bits
	HM_LastTicksStateRest:ULINT;						//System ticks value last time left rest state
	HM_Empty:BOOL;										//Flag machinpart is empty
	HM_MtrRevDone:bool;									//Flag motors ran in reverse
	HM_CamReceivedData: ARRAY[0..100] OF BYTE;			//Received data from camera
	HM_CamOmronFhEthReceivedData: STRING;				//Received data from omron FhEth controller
	
	DataBuilder:utl_Any_DataBuilder;
	HM_InfoString:STRING;
	HM_DebugMultiStep_ResetInActivations:BOOL;			//enable testing if multistep works correctly
	HM_DebugServoRestart:bool;
	
